IF (MaquinaModoManual) THEN
	//Controle Manual - Válvula Y4
	IF (IhmBt_Y4_Ligar) THEN
		OutValvulaY4R := FALSE;	//Solenóide de Recuo
		OutValvulaY4A := TRUE; //Solenóide de Avanço
	ELSE
		OutValvulaY4A := FALSE;	//Solenóide de Avanço
		OutValvulaY4R := TRUE; //Solenóide de Recuo	
	END_IF
ELSIF (MaquinaModoAuto) THEN
	//Controle Automático - Válvula Y4
	IF (AvancarValvulaY4) THEN
		OutValvulaY4R := FALSE; //Solenóide de Recuo
		OutValvulaY4A := TRUE;	//Solenóide de Avanço
	ELSE
		OutValvulaY4A := FALSE; //Solenóide de Avanço
		OutValvulaY4R := TRUE;	//Solenóide de Recuo
	END_IF
ELSE
	OutValvulaY4R := FALSE; //Solenóide de Recuo
	OutValvulaY4A := FALSE;	//Solenóide de Avanço
END_IF

(*========================================================================*)

(*==============		Válvula Y5 - XXXXXXX XXXXXXX		==============*)

IF (MaquinaModoManual) THEN
	//Controle Manual - Válvula Y5
	IF (IhmBt_Y5_Ligar) THEN
		OutValvulaY5R := FALSE;	//Solenóide de Recuo
		OutValvulaY5A := TRUE; //Solenóide de Avanço
	ELSE
		OutValvulaY5A := FALSE;	//Solenóide de Avanço
		OutValvulaY5R := TRUE; //Solenóide de Recuo	
	END_IF
ELSIF (MaquinaModoAuto) THEN
	//Controle Automático - Válvula Y5
	IF (AvancarValvulaY5) THEN
		OutValvulaY5R := FALSE; //Solenóide de Recuo
		OutValvulaY5A := TRUE;	//Solenóide de Avanço
	ELSE
		OutValvulaY5A := FALSE; //Solenóide de Avanço
		OutValvulaY5R := TRUE;	//Solenóide de Recuo
	END_IF
ELSE
	OutValvulaY5R := FALSE; //Solenóide de Recuo
	OutValvulaY5A := FALSE;	//Solenóide de Avanço
END_IF

(*========================================================================*)

(*==============		Válvula Y6 - XXXXXXX XXXXXXX		==============*)

IF (MaquinaModoManual) THEN
	//Controle Manual - Válvula Y6
	IF (IhmBt_Y6_Ligar) THEN
		OutValvulaY6 := TRUE;
	ELSE
		OutValvulaY6 := FALSE;
	END_IF
ELSIF (MaquinaModoAuto) THEN
	//Controle Automático - Válvula Y6
	IF (LigarValvulaY6) THEN
		OutValvulaY6 := TRUE;
	ELSE
		OutValvulaY6 := FALSE;
	END_IF
ELSE
	OutValvulaY6 := FALSE;
END_IF

(*========================================================================*)

(*==============		Válvula Y9 - XXXXXXX XXXXXXX		==============*)

IF (MaquinaModoManual) THEN
	//Controle Manual - Válvula Y9
	IF (IhmBt_Y9_Ligar) THEN
		OutValvulaY9 := TRUE;
	ELSE
		OutValvulaY9 := FALSE;
	END_IF
ELSIF (MaquinaModoAuto) THEN
	//Controle Automático - Válvula Y9
	IF (LigarValvulaY9) THEN
		OutValvulaY9 := TRUE;
	ELSE
		OutValvulaY9 := FALSE;
	END_IF
ELSE
	OutValvulaY9 := FALSE;
END_IF

(*========================================================================*)

(*==========		Válvula Proporcional - XXXXXXX XXXXXXX		==========*)

IF (MaquinaModoManual) THEN
	//Controle Manual - Válvula Proporcional
	IF (IhmBt_VP_Teste) THEN
		ValvulaProporcional := (INT_TO_REAL(IhmEscr_ValvulaProporcional)/100)*(32767);
	END_IF
ELSIF (MaquinaModoAuto) THEN
	//Controle Automático - Válvula Proporcional
	ValvulaProporcional := (INT_TO_REAL(50)/100)*(32767);
ELSE
	ValvulaProporcional := 0;
END_IF
	
(*========================================================================*)

(*=============		Válvula Y7 - Válvula de Segurança 1		==============*)

//Controle Automático - Válvula Y7
IF (NOT Alarmes.AlarmeGrave) THEN
	LigarValvulaY7 := TRUE;
ELSE
	LigarValvulaY7 := FALSE;
END_IF

//Válvula Y7 - XXXXX XXXXX
IF (LigarValvulaY7) THEN
	OutValvulaY7 := TRUE;
ELSE
	OutValvulaY7 := FALSE;
END_IF

(*========================================================================*) 

(*=============		Válvula Y8 - Válvula de Segurança 2		==============*)

//Controle Automático - Válvula Y8
IF (NOT Alarmes.AlarmeGrave) THEN
	LigarValvulaY8 := TRUE;
ELSE
	LigarValvulaY8 := FALSE;
END_IF

//Válvula Y8 - XXXXX XXXXX
IF (LigarValvulaY8) THEN
	OutValvulaY8 := TRUE;
ELSE
	OutValvulaY8 := FALSE;
END_IF

(*========================================================================*)

END_PROGRAM

// ---- POUs/Perifericos/ReguaPotenciometrica.TcPOU
PROGRAM ReguaPotenciometrica
VAR
	
(*==================		RÉGUA POTENCIOMÉTRICA		==================*)	
 

 
(*========================================================================*)

END_VAR

(*==========		Régua Potênciométrica - EL3004 - 15 bits	==========*)

ReguaPotenciometricaPosicao := (INT_TO_REAL(ReguaPotenciometricaSinal)/32787)*100;

(*=========================		Calibração		==========================*)

IF (MaquinaModoManual) THEN

	IF (IhmBt_ReguaPotenciometrica_CalibrarRecuo) THEN
		ReguaPotenciometrica_Recuada := (INT_TO_REAL(ReguaPotenciometricaSinal)/32787)*100;
		ReguaPotenciometrica_Recuada_LI := (1-(IhmEscr_ReguaPotenciometrica_ToleranciaRecuo/100))*ReguaPotenciometrica_Recuada;
		ReguaPotenciometrica_Recuada_LS := (1+(IhmEscr_ReguaPotenciometrica_ToleranciaRecuo/100))*ReguaPotenciometrica_Recuada;
	END_IF
	
	IF (IhmBt_ReguaPotenciometrica_CalibrarPorca) THEN
		ReguaPotenciometrica_Porca := (INT_TO_REAL(ReguaPotenciometricaSinal)/32787)*100;
		ReguaPotenciometrica_Porca_LI := (1-(IhmEscr_ReguaPotenciometrica_ToleranciaPorca/100))*ReguaPotenciometrica_Porca;
		ReguaPotenciometrica_Porca_LS := (1+(IhmEscr_ReguaPotenciometrica_ToleranciaPorca/100))*ReguaPotenciometrica_Porca;
	END_IF
	
	IF (IhmBt_ReguaPotenciometrica_CalibrarAvanco) THEN
		ReguaPotenciometrica_Avancada := (INT_TO_REAL(ReguaPotenciometricaSinal)/32787)*100;
		ReguaPotenciometrica_Avancada_LI := (1-(IhmEscr_ReguaPotenciometrica_ToleranciaAvanco/100))*ReguaPotenciometrica_Avancada;
		ReguaPotenciometrica_Avancada_LS := (1+(IhmEscr_ReguaPotenciometrica_ToleranciaAvanco/100))*ReguaPotenciometrica_Avancada;
	END_IF
	
END_IF

(*======================		Modo Automático		======================*)


(*========================================================================*)

END_PROGRAM

// ---- POUs/Perifericos/Servos.TcPOU
PROGRAM Servos
VAR
	DelayTeste				: TON;
	
	VetorPosicaoX	: ARRAY[0..15] OF LREAL;
	VetorPosicaoY	: ARRAY[0..15] OF LREAL;
	
	Delay_BtReferenciarServoX 	: TON;
	Delay_BtReferenciarServoY 	: TON;
	
	ServoX_Referenciar			: BOOL;
	ServoY_Referenciar			: BOOL;
	
	ServoX_ReferenciarAuto		: BOOL;
	ServoY_ReferenciarAuto		: BOOL;
	
(*==========================		POWER		==========================*)	

	EixoX_Power 			: MC_Power;	
	EixoX_Power_Busy		: BOOL;
	EixoX_Power_Active		: BOOL;
	EixoX_Power_Error		: BOOL;
	EixoX_Power_ErrorID		: UDINT;
	
	EixoY_Power 			: MC_Power;	
	EixoY_Power_Busy		: BOOL;
	EixoY_Power_Active		: BOOL;
	EixoY_Power_Error		: BOOL;
	EixoY_Power_ErrorID		: UDINT;

(*========================================================================*)

(*==========================		RESET		==========================*)	

	EixoX_Reset 			: MC_Reset;
	EixoX_Reset_Done		: BOOL;	
	EixoX_Reset_Busy		: BOOL;
	EixoX_Reset_Error		: BOOL;
	EixoX_Reset_ErrorID		: UDINT;
	
	EixoY_Reset 			: MC_Reset;
	EixoY_Reset_Done		: BOOL;	
	EixoY_Reset_Busy		: BOOL;
	Eixoy_Reset_Error		: BOOL;
	EixoY_Reset_ErrorID		: UDINT;

(*========================================================================*)

(*==========================		HOME		==========================*)	

	EixoX_Home 						: MC_Home;
	EixoX_Home_Done					: BOOL;	
	EixoX_Home_CommandAborted		: BOOL;
	EixoX_Home_Error				: BOOL;
	EixoX_Home_ErrorID				: UDINT;
	
	HomingMode     					: MC_HomingMode;
	
	EixoY_Home 						: MC_Home;
	EixoY_Home_Done					: BOOL;	
	EixoY_Home_CommandAborted		: BOOL;
	EixoY_Home_Error				: BOOL;
	EixoY_Home_ErrorID				: UDINT;

(*========================================================================*)

(*======================		MOVE ABSOLUTE		======================*)	

	EixoX_MoveAbsHome					: MC_MoveAbsolute;
	EixoX_MoveAbsHome_Done				: BOOL;	
	EixoX_MoveAbsHome_CommandAborted	: BOOL;
	EixoX_MoveAbsHome_Error				: BOOL;
	EixoX_MoveAbsHome_ErrorID			: UDINT;
	
	EixoY_MoveAbsHome					: MC_MoveAbsolute;
	EixoY_MoveAbsHome_Done				: BOOL;	
	EixoY_MoveAbsHome_CommandAborted	: BOOL;
	EixoY_MoveAbsHome_Error				: BOOL;
	EixoY_MoveAbsHome_ErrorID			: UDINT;

	EixoX_MoveAbsolute 					: MC_MoveAbsolute;
	EixoX_MoveAbsolute_Done				: BOOL;	
	EixoX_MoveAbsolute_CommandAborted	: BOOL;
	EixoX_MoveAbsolute_Error			: BOOL;
	EixoX_MoveAbsolute_ErrorID			: UDINT;
	
	EixoY_MoveAbsolute			 		: MC_MoveAbsolute;
	EixoY_MoveAbsolute_Done				: BOOL;	
	EixoY_MoveAbsolute_CommandAborted	: BOOL;
	EixoY_MoveAbsolute_Error			: BOOL;
	EixoY_MoveAbsolute_ErrorID			: UDINT;

(*========================================================================*)
	
(*=========================		MOVE JOG		==========================*)	

	EixoX_MoveJog					: MC_Jog;
	EixoY_MoveJog					: MC_Jog;
	
	EixoX_JogReferenciarAuto		: MC_Jog;
	EixoY_JogReferenciarAuto		: MC_Jog;
	
(*========================================================================*)	

(*======================		MOVE RELATIVE		======================*)	

	EixoX_MoveRelative		: MC_MoveRelative;
	EixoY_MoveRelative		: MC_MoveRelative;

(*========================================================================*)

(*=====================		MÁQUINA DE ESTADOS		======================*)	

	PassoServosXY				: INT;
	index						: INT;
	PosicaoX					: LREAL;
	PosicaoY					: LREAL;
	
	Flag_EixoX_PosicaoOK		: BOOL;
	Flag_EixoY_PosicaoOK		: BOOL;
	
	PassoEixoXReferenciarAutoINICIO	: INT;
	PassoEixoXReferenciarAutoFIM	: INT;
	PassoEixoYReferenciarAutoINICIO	: INT;
	PassoEixoYReferenciarAutoFIM	: INT;
	
	JogFwd_EixoX_ReferenciarAuto	: BOOL;
	JogBwd_EixoX_ReferenciarAuto	: BOOL;

	JogFwd_EixoY_ReferenciarAuto	: BOOL;
	JogBwd_EixoY_ReferenciarAuto	: BOOL;

(*========================================================================*)
	
	//Blocos de Controle Eixo X
	PowerOnServoX		: BOOL;
	ReferenciarServoX	: BOOL;
	MoveHomeServoX		: BOOL;
	ResetServoX			: BOOL;
	JogFwdServoX		: BOOL;
	JogBwdServoX		: BOOL;
	
	//Status Servo Eixo X
	VelocidadeEixoX		: LREAL;
	PosicaoEixoX		: LREAL;
	TorqueEixoX			: LREAL;
	
	//Blocos de Controle Eixo Y
	PowerOnServoY		: BOOL;
	ReferenciarServoY	: BOOL;
	MoveHomeServoY		: BOOL;
	ResetServoY			: BOOL;
	JogFwdServoY		: BOOL;
	JogBwdServoY		: BOOL;
	
	//Status Servo Eixo X
	VelocidadeEixoY		: LREAL;
	PosicaoEixoY		: LREAL;
	TorqueEixoY			: LREAL;
	
END_VAR

IhmEscr_ServoXY_VelocidadeManual := 5;

(*=================		POWER - SERVOS EIXOS X E Y		==================*)

(*======================		SERVO EIXO X		======================*)

EixoX_Power_Busy 	:= EixoX_Power.Busy;
EixoX_Power_Active 	:= EixoX_Power.Active;
EixoX_Power_Error 	:= EixoX_Power.Error;
EixoX_Power_ErrorID	:= EixoX_Power.ErrorID;

IF (MaquinaModoManual AND NOT Alarmes.AlarmeGrave)THEN
	EixoX_Power(Axis := EixoX,
				Enable := IhmBt_ServoX_PowerOn,
				Enable_Positive := IhmBt_ServoX_PowerOn,
				Enable_Negative := IhmBt_ServoX_PowerOn,
				Override := 100);
ELSIF (NOT Alarmes.AlarmeGrave) THEN
	EixoX_Power(Axis := EixoX,
			Enable := TRUE,
			Enable_Positive := TRUE,
			Enable_Negative := TRUE,
			Override := 100);
ELSE
	EixoX_Power(Axis := EixoX,
			Enable := FALSE,
			Enable_Positive := FALSE,
			Enable_Negative := FALSE);
END_IF
				
IF EixoX_Power.Status THEN
	EixoX_Energizado := TRUE;
ELSE
	EixoX_Energizado := FALSE;
END_IF

(*======================		SERVO EIXO Y		======================*)

EixoY_Power_Busy 	:= EixoY_Power.Busy;
EixoY_Power_Active 	:= EixoY_Power.Active;
EixoY_Power_Error 	:= EixoY_Power.Error;
EixoY_Power_ErrorID	:= EixoY_Power.ErrorID;

IF (MaquinaModoManual AND NOT Alarmes.AlarmeGrave)THEN
	EixoY_Power(Axis := EixoY,
				Enable := IhmBt_ServoY_PowerOn,
				Enable_Positive := IhmBt_ServoY_PowerOn,
				Enable_Negative := IhmBt_ServoY_PowerOn,
				Override := 100);
ELSIF (NOT Alarmes.AlarmeGrave) THEN
	EixoY_Power(Axis := EixoY,
			Enable := TRUE,
			Enable_Positive := TRUE,
			Enable_Negative := TRUE,
			Override := 100);
ELSE
	EixoY_Power(Axis := EixoY,
			Enable := FALSE,
			Enable_Positive := FALSE,
			Enable_Negative := FALSE);
END_IF
			
IF EixoY_Power.Status THEN
	EixoY_Energizado := TRUE;
ELSE
	EixoY_Energizado := FALSE;
END_IF

(*=================		RESET - SERVOS EIXOS X E Y		==================*)

(*======================		SERVO EIXO X		======================*)

EixoX_Reset_Done 	:= EixoX_Reset.Done;
EixoX_Reset_Busy 	:= EixoX_Reset.Busy;
EixoX_Reset_Error 	:= EixoX_Reset.Error;
EixoX_Reset_ErrorID	:= EixoX_Reset.ErrorID;

EixoX_Reset(Axis := EixoX, Execute := (IhmBt_ServoX_Reset OR Reset));

(*======================		SERVO EIXO Y		======================*)

EixoY_Reset_Done 	:= EixoY_Reset.Done;
EixoY_Reset_Busy 	:= EixoY_Reset.Busy;
EixoY_Reset_Error 	:= EixoY_Reset.Error;
EixoY_Reset_ErrorID	:= EixoY_Reset.ErrorID;

EixoY_Reset(Axis := EixoY, Execute := (IhmBt_ServoX_Reset OR Reset));

(*=============		REFERENCIAR - SERVOS EIXOS X E Y		==============*)

(*======================		SERVO EIXO X		======================*)

EixoX_Home_Done 			:= EixoX_Home.Done;
EixoX_Home_CommandAborted 	:= EixoX_Home.CommandAborted;
EixoX_Home_Error 			:= EixoX_Home.Error;
EixoX_Home_ErrorID			:= EixoX_Home.ErrorID;

//Lógica para Delay ao pressionar o botão de referenciar
	IF (IhmBt_ServoX_Referenciar) THEN
		Delay_BtReferenciarServoX(IN := TRUE, PT := T#2S);
		IF(Delay_BtReferenciarServoX.Q) THEN
			ServoX_Referenciar := TRUE;
		END_IF
	ELSE
		Delay_BtReferenciarServoX(IN := FALSE);
		ServoX_Referenciar := FALSE;
	END_IF

EixoX_Home(Axis := EixoX, Position := 0, HomingMode := MC_Direct, Execute := ((ServoX_Referenciar AND MaquinaModoManual) OR ServoX_ReferenciarAuto));

(*======================		SERVO EIXO Y		======================*)

EixoY_Home_Done 			:= EixoY_Home.Done;
EixoY_Home_CommandAborted 	:= EixoY_Home.CommandAborted;
EixoY_Home_Error 			:= EixoY_Home.Error;
EixoY_Home_ErrorID			:= EixoY_Home.ErrorID;

//Lógica para Delay ao pressionar o botão de referenciar
	IF (IhmBt_ServoY_Referenciar) THEN
		Delay_BtReferenciarServoY(IN := TRUE, PT := T#2S);
		IF(Delay_BtReferenciarServoY.Q) THEN
			ServoY_Referenciar := TRUE;
		END_IF
	ELSE
		Delay_BtReferenciarServoY(IN := FALSE);
		ServoY_Referenciar := FALSE;
	END_IF

EixoY_Home(Axis := EixoY, Position := 0, HomingMode := MC_Direct, Execute := ((ServoY_Referenciar AND MaquinaModoManual) OR ServoY_ReferenciarAuto));

(*=============		MOVE para HOME - SERVOS EIXOS X E Y		==============*)

(*======================		SERVO EIXO X		======================*)

EixoX_MoveAbsHome(	Axis := EixoX,
					Execute := (IhmBt_ServoX_Home AND MaquinaModoManual),
					Position := 0,
					Velocity := IhmEscr_ServoXY_VelocidadeAuto
					(*Direction := 2*));

(*======================		SERVO EIXO Y		======================*)
								
EixoX_MoveAbsHome(	Axis := EixoY,
					Execute := (IhmBt_ServoY_Home AND MaquinaModoManual),
					Position := 0,
					Velocity := IhmEscr_ServoXY_VelocidadeAuto
					(*Direction := 2*));

(*=================		MANUAL - SERVOS EIXOS X E Y		==================*)

(*======================		SERVO EIXO X		======================*)

EixoX_MoveJog(	Axis := EixoX,
				JogForward := (IhmBt_ServoX_JogFwd AND MaquinaModoManual),
				JogBackwards := (IhmBt_ServoX_JogBwd AND MaquinaModoManual),
				Velocity := IhmEscr_ServoXY_VelocidadeManual,
				Acceleration := 100,
				Deceleration := 100);
				
(*======================		SERVO EIXO Y		======================*)
								
EixoY_MoveJog(	Axis := EixoY,
				JogForward := (IhmBt_ServoY_JogFwd AND MaquinaModoManual),
				JogBackwards := (IhmBt_ServoY_JogBwd AND MaquinaModoManual),
				Velocity := IhmEscr_ServoXY_VelocidadeManual,
				Acceleration := 100,
				Deceleration := 100);

(*=================		STATUS - SERVOS EIXOS X E Y		==================*)

(*======================		SERVO EIXO X		======================*)

IhmLeit_ServoX_Posicao		:= EixoX.NcToPlc.ActPos;
IhmLeit_ServoX_Velocidade	:= EixoX.NcToPlc.ActVelo;
IhmLeit_ServoX_Torque		:= EixoX.NcToPlc.ActTorque;

(*======================		SERVO EIXO Y		======================*)

IhmLeit_ServoY_Posicao		:= EixoY.NcToPlc.ActPos;
IhmLeit_ServoY_Velocidade	:= EixoY.NcToPlc.ActVelo;
IhmLeit_ServoY_Torque		:= EixoY.NcToPlc.ActTorque;

(*=========		MANIVELA ELETRÔNICA - SERVOS EIXOS X E Y		==========*)



(*=================		AUTOMÁTICO - SERVOS EIXOS X E Y		==============*)
(*======================		Modo Automático		======================*)

//Receita Teste

PosicaoOrigemX := 20;
PosicaoOrigemY := 31;

VetorPosicaoX[0] := 20;
VetorPosicaoY[0] := 31;

VetorPosicaoX[1] := 59;
VetorPosicaoY[1] := 15;

//PosicaoOrigemX := TargetX[0];
//PosicaoOrigemY := TargetY[0];

//Condição de Bloqueio da Máquina de Estados - Servos XY
IF (Alarmes.AlarmeGrave
	//OR NOT Alarmes.AlarmeMedio
	OR NOT MaquinaLigada
	OR NOT MaquinaModoAuto
	//OR NOT((ReguaPotenciometricaPosicao > ReguaPotenciometrica_Recuada_LI) AND (ReguaPotenciometricaPosicao < ReguaPotenciometrica_Recuada_LS))
	) THEN
	PassoServosXY := 1000;
	Flag_ServosXY_Maquina := FALSE;
	index := 0;
	EixoX_MoveAbsolute(	Axis:= EixoX, Execute:= FALSE);
	EixoY_MoveAbsolute(	Axis:= EixoY, Execute:= FALSE);
	Flag_EixoX_PosicaoOK := FALSE;
	Flag_EixoY_PosicaoOK := FALSE;
	
END_IF

CASE PassoServosXY OF
	
	//Passo 0 - Inicialização	
	0: PassoServosXY := 10;
		
	//Passo 10 - Condição para Iniciar a Rotina dos Servos XY
	10: IF  (Flag_Maquina_ServosXY) THEN
			Flag_Maquina_ServosXY := FALSE;
			PassoServosXY := 20;
		END_IF
		
	//Passo 20 - Soldar 
	20:	IF (TRUE OR SoldaXY[index]) THEN
			Flag_ServosXY_MaquinaSolda := TRUE;
			PassoServosXY := 30;
		ELSE
			Flag_ServosXY_MaquinaSolda := FALSE;
			PassoServosXY := 40;			
		END_IF

	//Passo 30 - Aguardar conclusão de Solda
	30:	IF (Flag_MaquinaSolda_ServosXY) THEN
			Flag_MaquinaSolda_ServosXY := FALSE;
			PassoServosXY := 40;			
		END_IF
	
	//Passo 40 - Validar Próximo Ponto (X,Y)
	40: index := index + 1;
		IF (index<=(NumPontosSolda-1)) THEN
			PassoServosXY := 50;	
		ELSE
			index := 0;
			PassoServosXY := 80;	
		END_IF
	
	//Passo 50 - Carregar Posição Alvo - Servo X e Y 
	50: PosicaoX := VetorPosicaoX[index];//TargetX[index];
		PosicaoY := VetorPosicaoY[index];//TargetY[index];
		PassoServosXY := 60;
		
	//Passo 60 - Movimentar Servo Eixos X e Y
	//			aguardar conclusão do movimento
	60: EixoX_MoveAbsolute(	Axis:= EixoX, 
							Execute:= TRUE,
							Position:= PosicaoX,
							Velocity:= IhmEscr_ServoXY_VelocidadeAuto
							//Acceleration:= 15000,
							//Deceleration:= 15000
							);			
		IF (EixoX_MoveAbsolute.Done) THEN
			Flag_EixoX_PosicaoOK := TRUE;
		END_IF
							
		EixoY_MoveAbsolute(	Axis:= EixoY, 
							Execute:= TRUE,
							Position:= PosicaoY,
							Velocity:= IhmEscr_ServoXY_VelocidadeAuto
							//Acceleration:= 15000,
							//Deceleration:= 15000
							);
		IF (EixoY_MoveAbsolute.Done) THEN
			Flag_EixoY_PosicaoOK := TRUE;	
		END_IF
		
		IF (Flag_EixoX_PosicaoOK AND Flag_EixoY_PosicaoOK) THEN
			PassoServosXY := 70;	
		END_IF
		
	//Passo 70 - Finalizar Movimentação - Servos X e Y
	70: EixoX_MoveAbsolute(	Axis:= EixoX, Execute:= FALSE);
		EixoY_MoveAbsolute(	Axis:= EixoY, Execute:= FALSE);
		Flag_EixoX_PosicaoOK := FALSE;
		Flag_EixoY_PosicaoOK := FALSE;
		PassoServosXY := 75;
		
	//Passo 75 - Aguardar Delay de Teste
	75: DelayTeste(IN:=TRUE,PT:=T#200MS);
		IF DelayTeste.Q THEN
			DelayTeste(IN:=FALSE);
			PassoServosXY := 20;		
		END_IF
		
	//Passo 80 - Movimentar Servos X e  para a Origem
	//			e aguardar conclusão do movimento
	80: EixoX_MoveAbsolute(	Axis := EixoX, 
							Execute := TRUE,
							Position := VetorPosicaoX[0],
							Velocity := IhmEscr_ServoXY_VelocidadeAuto
							//Acceleration:= 15000,
							//Deceleration:= 15000
							);
		IF (EixoX_MoveAbsolute.Done) THEN
			Flag_EixoX_PosicaoOK := TRUE;	
		END_IF
		
		EixoY_MoveAbsolute(	Axis := EixoY, 
							Execute := TRUE,
							Position := VetorPosicaoY[0],
							Velocity := IhmEscr_ServoXY_VelocidadeAuto
							//Acceleration:= 15000,
							//Deceleration:= 15000
							);
		IF (EixoY_MoveAbsolute.Done) THEN
			Flag_EixoY_PosicaoOK := TRUE;	
		END_IF
		
		IF (Flag_EixoX_PosicaoOK AND Flag_EixoY_PosicaoOK) THEN
			PassoServosXY := 90;	
		END_IF
		
	//Passo 90 - Finalizar Movimentação - Servos X e Y
	90: EixoX_MoveAbsolute(	Axis:= EixoX, Execute:= FALSE);
		EixoY_MoveAbsolute(	Axis:= EixoY, Execute:= FALSE);
		Flag_EixoX_PosicaoOK := FALSE;
		Flag_EixoY_PosicaoOK := FALSE;
		PassoServosXY := 100;
		
	//Passo 100 - Sinalizar Conclusão da Rotina
	100:	Flag_ServosXY_Maquina := TRUE;
		PassoServosXY := 1000;

	//Passo 1000 - Finalização
	1000: PassoServosXY := 0;
	
END_CASE

(*=================		REFERENCIAMENTO AUTOMÁTICO		==================*)

(*======================		SERVO EIXO X		======================*)
								
EixoX_JogReferenciarAuto(	Axis := EixoX,
							JogForward := (JogFwd_EixoX_ReferenciarAuto),
							JogBackwards := (JogBwd_EixoX_ReferenciarAuto),
							Velocity := 1,
							Acceleration := 100,
							Deceleration := 100);
							
//Condição de Bloqueio da Máquina de Estados - Referenciamento Auto (INICIO)
IF (Alarmes.AlarmeGrave
	OR MaquinaLigada
	OR NOT MaquinaModoManual
	OR NOT IhmBt_ServoX_ReferenciarAutoINICIO
	OR	IhmBt_ServoX_ReferenciarAutoFIM
	OR NOT IhmBt_ServoX_PowerOn
	OR InFimCurso3
	) THEN
	PassoEixoXReferenciarAutoINICIO := 1000;
	//JogFwd_EixoX_ReferenciarAuto := FALSE;
	JogBwd_EixoX_ReferenciarAuto := FALSE;
	//ServoX_ReferenciarAuto := FALSE;
END_IF

CASE PassoEixoXReferenciarAutoINICIO OF

	//Passo 0 - Inicialização
	0: PassoEixoXReferenciarAutoINICIO := 10;
	
	//Passo 10 - Condição para iniciar Rotina de Referenciamento Automático
	10: IF (IhmBt_ServoX_ReferenciarAutoINICIO) THEN
			PassoEixoXReferenciarAutoINICIO := 20;
		END_IF
		
	//Passo 20 - Move Jog BWD - Referenciar 
	20: JogBwd_EixoX_ReferenciarAuto := TRUE;
		PassoEixoXReferenciarAutoINICIO := 30;

	//Passo 30 - Aguardar Acionamento do Switch Fim de Curso
	30: IF (InFimCurso3) THEN
			JogBwd_EixoX_ReferenciarAuto := TRUE;
			//ServoX_ReferenciarAuto := TRUE;
			PassoEixoXReferenciarAutoINICIO := 40;
		END_IF
		
	//Passo 40 - Sinalizar Conclusão da Rotina
	40: IhmBt_ServoX_ReferenciarAutoINICIO := FALSE;
		//ServoX_ReferenciarAuto := FALSE;
		PassoEixoXReferenciarAutoINICIO := 1000;
	
	//Passo 1000 - Finalização
	1000:	IhmBt_ServoX_ReferenciarAutoINICIO := FALSE;
			PassoEixoXReferenciarAutoINICIO := 0;

END_CASE

//Condição de Bloqueio da Máquina de Estados - Referenciamento Auto (FIM)
IF (Alarmes.AlarmeGrave
	OR MaquinaLigada
	OR NOT MaquinaModoManual
	OR NOT IhmBt_ServoX_ReferenciarAutoFIM
	OR IhmBt_ServoX_ReferenciarAutoINICIO
	OR NOT IhmBt_ServoX_PowerOn
	OR InFimCurso4
	) THEN
	PassoEixoXReferenciarAutoFIM := 1000;
	JogFwd_EixoX_ReferenciarAuto := FALSE;
	//JogBwd_EixoX_ReferenciarAuto := FALSE;
	//ServoX_ReferenciarAuto := FALSE;
END_IF

CASE PassoEixoXReferenciarAutoFIM OF

	//Passo 0 - Inicialização
	0: PassoEixoXReferenciarAutoFIM := 10;
	
	//Passo 10 - Condição para iniciar Rotina de Referenciamento Automático
	10: IF (IhmBt_ServoX_ReferenciarAutoFIM) THEN
			PassoEixoXReferenciarAutoFIM := 20;
		END_IF
		
	//Passo 20 - Move Jog FWD - Referenciar 
	20: JogFwd_EixoX_ReferenciarAuto := TRUE;
		PassoEixoXReferenciarAutoFIM := 30;

	//Passo 30 - Aguardar Acionamento do Switch Fim de Curso
	30: IF (InFimCurso4) THEN
			JogFwd_EixoX_ReferenciarAuto := TRUE;
			//ServoX_ReferenciarAuto := TRUE;
			PassoEixoXReferenciarAutoFIM := 40;
		END_IF
		
	//Passo 40 - Sinalizar Conclusão da Rotina
	40: IhmBt_ServoX_ReferenciarAutoFIM := FALSE;
		//ServoX_ReferenciarAuto := FALSE;
		PassoEixoXReferenciarAutoFIM := 1000;
	
	//Passo 1000 - Finalização
	1000:	IhmBt_ServoX_ReferenciarAutoFIM := FALSE;
			PassoEixoXReferenciarAutoFIM := 0;

END_CASE

(*======================		SERVO EIXO Y		======================*)
								
EixoY_JogReferenciarAuto(	Axis := EixoY,
							JogForward := (JogFwd_EixoY_ReferenciarAuto),
							JogBackwards := (JogBwd_EixoY_ReferenciarAuto),
							Velocity := 1,
							Acceleration := 100,
							Deceleration := 100);
							
//Condição de Bloqueio da Máquina de Estados - Referenciamento Auto (INICIO)
IF (Alarmes.AlarmeGrave
	OR MaquinaLigada
	OR NOT MaquinaModoManual
	OR NOT IhmBt_ServoY_ReferenciarAutoINICIO
	OR IhmBt_ServoY_ReferenciarAutoFIM
	OR NOT IhmBt_ServoY_PowerOn
	OR InFimCurso1
	) THEN
	PassoEixoYReferenciarAutoINICIO := 1000;
	//JogFwd_EixoY_ReferenciarAuto := FALSE;
	JogBwd_EixoY_ReferenciarAuto := FALSE;
	//ServoY_ReferenciarAuto := FALSE;
END_IF

CASE PassoEixoYReferenciarAutoINICIO OF

	//Passo 0 - Inicialização
	0: PassoEixoYReferenciarAutoINICIO := 10;
	
	//Passo 10 - Condição para iniciar Rotina de Referenciamento Automático
	10: IF (IhmBt_ServoY_ReferenciarAutoINICIO) THEN
			PassoEixoYReferenciarAutoINICIO := 20;
		END_IF
		
	//Passo 20 - Move Jog BWD - Referenciar 
	20: JogBwd_EixoY_ReferenciarAuto := TRUE;
		PassoEixoYReferenciarAutoINICIO := 30;

	//Passo 30 - Aguardar Acionamento do Switch Fim de Curso
	30: IF (InFimCurso1) THEN
			JogBwd_EixoY_ReferenciarAuto := TRUE;
			//ServoY_ReferenciarAuto := TRUE;
			PassoEixoYReferenciarAutoINICIO := 40;
		END_IF
		
	//Passo 40 - Sinalizar Conclusão da Rotina
	40: IhmBt_ServoY_ReferenciarAutoINICIO := FALSE;
		//ServoY_ReferenciarAuto := FALSE;
		PassoEixoYReferenciarAutoINICIO := 1000;
	
	//Passo 1000 - Finalização
	1000:	IhmBt_ServoY_ReferenciarAutoINICIO := FALSE;
			PassoEixoYReferenciarAutoINICIO := 0;

END_CASE

//Condição de Bloqueio da Máquina de Estados - Referenciamento Auto (FIM)
IF (Alarmes.AlarmeGrave
	OR MaquinaLigada
	OR NOT MaquinaModoManual
	OR NOT IhmBt_ServoY_ReferenciarAutoFIM
	OR IhmBt_ServoY_ReferenciarAutoINICIO
	OR NOT IhmBt_ServoY_PowerOn
	OR InFimCurso2
	) THEN
	PassoEixoYReferenciarAutoFIM := 1000;
	JogFwd_EixoY_ReferenciarAuto := FALSE;
	//JogBwd_EixoY_ReferenciarAuto := FALSE;
	//ServoY_ReferenciarAuto := FALSE;
END_IF

CASE PassoEixoYReferenciarAutoFIM OF

	//Passo 0 - Inicialização
	0: PassoEixoYReferenciarAutoFIM := 10;
	
	//Passo 10 - Condição para iniciar Rotina de Referenciamento Automático
	10: IF (IhmBt_ServoY_ReferenciarAutoFIM) THEN
			PassoEixoYReferenciarAutoFIM := 20;
		END_IF
		
	//Passo 20 - Move Jog FWD - Referenciar 
	20: JogBwd_EixoY_ReferenciarAuto := TRUE;
		PassoEixoYReferenciarAutoFIM := 30;

	//Passo 30 - Aguardar Acionamento do Switch Fim de Curso
	30: IF (InFimCurso1) THEN
			JogBwd_EixoY_ReferenciarAuto := TRUE;
			//ServoY_ReferenciarAuto := TRUE;
			PassoEixoYReferenciarAutoFIM := 40;
		END_IF
		
	//Passo 40 - Sinalizar Conclusão da Rotina
	40: IhmBt_ServoY_ReferenciarAutoFIM := FALSE;
		//ServoY_ReferenciarAuto := FALSE;
		PassoEixoYReferenciarAutoFIM := 1000;
	
	//Passo 1000 - Finalização
	1000:	IhmBt_ServoY_ReferenciarAutoFIM := FALSE;
			PassoEixoYReferenciarAutoFIM := 0;

END_CASE

(*========================================================================*)

END_PROGRAM

// ---- POUs/Perifericos/Robo.TcPOU
PROGRAM Robo
VAR

	BT_test						: BOOL;
	TON_DelayTesteExpPeca		: TON;
	
	//index						: INT;

(*=====================		ROBO YASKAWA		==========================*)	
 
 PassoRoboAuto				: INT;
 
 Flag_PLC_Robot_WorkHome		: BOOL; //Retonar a para a posição WORK HOME (Ordem PLC)
 Flag_PLC_Robot_PegarPeca		: BOOL; //Pegar Peça na Mesa Indexadora (Ordem PLC)
 Flag_PLC_Robot_Camera			: BOOL; //Levar Peça Até a Câmera (Ordem PLC)
 Flag_PLC_Robot_CapturarImagens	: BOOL;
 Flag_PLC_Robot_Aprovada		: BOOL; //Levar Peça Até a Caixa - Aprovada (Ordem PLC)
 Flag_PLC_Robot_Reprovada		: BOOL; //Descartar Peça (Ordem PLC)
 
 Flag_Robot_PLC_WorkHome		: BOOL; //Retonar a para a posição WORK HOME (Conclusão Robô)
 Flag_Robot_PLC_PegarPeca		: BOOL; //Pegar Peça na Mesa Indexadora (Conclusão Robô)
 Flag_Robot_PLC_Camera			: BOOL; //Levar Peça Até a Câmera (Conclusão Robô)
 Flag_Robot_PLC_CapturarImagens	: BOOL;
 Flag_Robot_PLC_Aprovada		: BOOL; //Levar Peça Até a Caixa - Aprovada (Conclusão Robô)
 Flag_Robot_PLC_Reprovada		: BOOL; //Descartar Peça (Conclusão Robô)

(*========================================================================*)

END_VAR

(*==========		Robô Yaskawa Comunicação Ethernet/IP		==========*)

//PLC to Robot -> Byte 0

PLC_Robot_0.0 := Robot_CallMasterJob;
PLC_Robot_0.1 := Robot_ServoOn;
PLC_Robot_0.2 := Robot_ServoOff;
PLC_Robot_0.3 := Robot_ExtStart;
PLC_Robot_0.4 := Robot_ResetAlarm;

//PLC_Robot_0.4 := Robot_JobBegin;

//PLC to Robot -> Byte 1

PLC_Robot_1.0 := Robot_JobCamera;

//PLC to Robot -> Byte 2

PLC_Robot_3 := 1; //Receita



Robot_NotSafetyPosition := Robot_PLC_0.3;
Robot_JobCompleted := Robot_PLC_1.0;

//Robot_Home:= Robot_PLC_1.0;

Robot_Peca	:= Robot_PLC_2.0;
Robot_Foto1	:= Robot_PLC_2.1;
Robot_Foto2	:= Robot_PLC_2.2;


Robot_HomePosition 	:= Robot_PLC_1.0;
Robot_TopMasterJob	:= Robot_PLC_1.1;
Robot_AlarmStatus 	:= Robot_PLC_1.2;




Robot_JobCamera := TRUE;

//Robot_PLC_1.0 := Valvula


(*=========================		Modo Manual		==========================*)

 PLC_Robot_2.0 := Flag_PLC_Robot_PegarPeca;
 PLC_Robot_2.1 := Flag_PLC_Robot_Camera;
 PLC_Robot_2.2 := Flag_PLC_Robot_CapturarImagens;
 PLC_Robot_2.3 := Flag_PLC_Robot_Aprovada;
 PLC_Robot_2.4 := Flag_PLC_Robot_Reprovada;
 PLC_Robot_2.5 := Flag_PLC_Robot_WorkHome;
 
 Flag_Robot_PLC_PegarPeca 		:= Robot_PLC_2.0;
 Flag_Robot_PLC_Camera 			:= Robot_PLC_2.1;
 Flag_Robot_PLC_CapturarImagens := Robot_PLC_2.2;
 Flag_Robot_PLC_Aprovada 		:= Robot_PLC_2.3;
 Flag_Robot_PLC_Reprovada 		:= Robot_PLC_2.4;
 Flag_Robot_PLC_WorkHome 		:= Robot_PLC_2.5;
 
(*======================		Modo Automático		======================*)

//Condição de Bloqueio da Máquina de Estados - Robô Yaskawa
IF (Alarmes.AlarmeGrave
	//OR NOT Alarmes.AlarmeMedio
	//OR NOT MaquinaLigada
	//OR NOT MaquinaModoAuto
	) THEN
	PassoRoboAuto := 1000;
	Camera_indexJob := 0;
END_IF

CASE PassoRoboAuto OF
	
	//Passo 0 - Inicialização	
	0: PassoRoboAuto := 10;
	   
	//Passo 10 - Condição para Iniciar a Rotina do Robo
	10: IF (Flag_Maquina_Robo) THEN
				Flag_Maquina_Robo := FALSE;
			PassoRoboAuto := 20;
		END_IF
		
	//Passo 20 - Verifica Posição do Robo
	20: IF (Robot_HomePosition) THEN
			PassoRoboAuto := 30;
		END_IF
		
	//Passo 30 - Verificar Flag Posição
	30:	IF (Flag_Robot_PLC_WorkHome) THEN
			PassoRoboAuto := 40;
		END_IF
			
	//Passo 40 - Iniciar Ciclo - Pegar Peça no Mesa Index
	40: Flag_PLC_Robot_PegarPeca := TRUE;
		IF (Flag_Robot_PLC_PegarPeca) THEN
			Flag_PLC_Robot_PegarPeca := FALSE;
			PassoRoboAuto := 50;	
		END_IF
		
	//Passo 50 - Levar Peça até a Câmera SICK 
	50: Flag_PLC_Robot_Camera := TRUE;
		IF (Flag_Robot_PLC_Camera) THEN
			Flag_PLC_Robot_Camera := FALSE;
			PassoRoboAuto := 60;	
		END_IF
			
	//Passo 60 - Sinalizar Captura de Imagens
	60: Flag_PLC_Robot_CapturarImagens := TRUE;
		IF (NOT Flag_Robot_PLC_Camera) THEN
			Flag_PLC_Robot_CapturarImagens := FALSE;
			PassoRoboAuto := 70;	
		END_IF
		
	//Passo 70 - Capturar Imagens
	70: Flag_Robo_Camera := TRUE;
		PassoRoboAuto := 80;
	
	//Passo 80 - Aguardar Conclusão da Capturar Imagens
	80: IF (Flag_Camera_Robo) THEN
			Flag_Camera_Robo := FALSE;
			PassoRoboAuto := 90;	
		END_IF	
			
	//Passo 90 - Avaliar Resultado da Câmera
	90: IF(PecaAprovada) THEN
			PecaAprovada := FALSE;
			PassoRoboAuto := 100;
		ELSE
			Camera_indexJob := 0;
			PassoRoboAuto := 120;
		END_IF

	//Passo 100 - Validar próximo ponto	
	100: IF (Camera_indexJob + 1 < NumPontosCamera) THEN
			Camera_indexJob := Camera_indexJob + 1;
			PassoRoboAuto := 50;
		ELSE
			Camera_indexJob := 0;
			PassoRoboAuto := 100;
		END_IF
	
	
	//Passo 100 - Depositar a Peça Aprovada na Caixa 
	110: Flag_PLC_Robot_Aprovada := TRUE;
		IF (Flag_Robot_PLC_Aprovada) THEN
			Flag_PLC_Robot_Aprovada := FALSE;
			
			//Expelir Peça da Garra
			AvancarValvulaY1 := TRUE;
			TON_DelayTesteExpPeca(IN := TRUE, PT := T#3S);
			IF (TON_DelayTesteExpPeca.Q) THEN
				TON_DelayTesteExpPeca(IN := FALSE);
				AvancarValvulaY1 := FALSE;
				PassoRoboAuto := 115;	
			END_IF

		END_IF
	
	//Passo 115 - Atualizar Contador de Peças Aprovadas
	115: Contador_PecasAprovadas := Contador_PecasAprovadas + 1;
		PassoRoboAuto := 130; 
		
	//Passo 120 - Descartar a Peça Reprovada 
	120: Flag_PLC_Robot_Reprovada := TRUE;
		IF (Flag_Robot_PLC_Reprovada) THEN
			Flag_PLC_Robot_Reprovada := FALSE;
			
			//Expelir Peça da Garra
			AvancarValvulaY1 := TRUE;
			TON_DelayTesteExpPeca(IN := TRUE, PT := T#3S);
			IF (TON_DelayTesteExpPeca.Q) THEN
				TON_DelayTesteExpPeca(IN := FALSE);
				AvancarValvulaY1 := FALSE;
				PassoRoboAuto := 125;
			END_IF
			
		END_IF
		
	//Passo 125 - Atualizar Contador de Peças Reprovadas
	125: Contador_PecasReprovadas := Contador_PecasReprovadas + 1;
		PassoRoboAuto := 130; 
	
	//Passo 130 - Atualizar Contador Total
	130: Contador_Total := Contador_PecasAprovadas + Contador_PecasReprovadas;
		PassoRoboAuto := 140; 
	
	//Passo 140 - Retornar a Posição WORK HOME 
	140: Flag_PLC_Robot_WorkHome := TRUE;
		IF (Flag_Robot_PLC_WorkHome) THEN
			Flag_PLC_Robot_WorkHome := FALSE;
			PassoRoboAuto := 150;	
		END_IF
		
	//Passo 150 - Sinalizar Conclusão da Rotina 
	150: Flag_Robo_Maquina := TRUE;
		PassoRoboAuto := 1000;

	//Passo 1000 - Finalização
	1000: PassoRoboAuto := 0;
	
END_CASE

(*========================================================================*)

END_PROGRAM

// ---- POUs/Perifericos/Camera.TcPOU
PROGRAM Camera
VAR

	BT_test						: BOOL;
	
	TON_DelayTest1				: TON;
	TON_DelayTest2				: TON;
	TON_DelayTest3				: TON;
	TON_DelayTest4				: TON;
	TON_DelayTest5				: TON;

(*=========================		CAMERA SICK		==========================*)	
 
 PassoCameraAuto			: INT;
 TON_CameraError			: TON;
 TON_CameraChangeJob		: TON;
 
(*========================================================================*)

END_VAR

(*=============		Câmera Sick Comunicação Ethernet/IP		==============*)

Camera_JobResult := CameraSickIn_3.0;
Camera_JobCompleted := CameraSickIn_0.2;
Camera_JobID := CameraSickIn_2;

CameraSickOut_0.0 := Camera_Trigger;
CameraSickOut_0.1 := Camera_ChangeJob;
CameraSickOut_2 := Camera_SetJob;

(*========================================================================*)

IhmLeit_Camera_JobID := BYTE_TO_INT(Camera_JobID);

IhmVs_Camera_JobResult_Text := 'Test';

(*=========================		Modo Manual		==========================*)

IF (MaquinaModoManual) THEN

	Camera_SetJob := INT_TO_BYTE(IhmEscr_Camera_SetJob);
	Camera_ChangeJob := IhmBt_Camera_ChangeJob;
	Camera_Trigger := IhmBt_Camera_Trigger;

END_IF

(*======================		Modo Automático		======================*)

Camera_TargetJob[0] := 1;
Camera_TargetJob[1] := 2;

//Condição de Bloqueio da Máquina de Estados - Câmera SICK
IF (Alarmes.AlarmeGrave
	//OR NOT Alarmes.AlarmeMedio
	//OR NOT MaquinaLigada
	OR NOT MaquinaModoAuto
	) THEN
	PassoCameraAuto := 1000;
END_IF

CASE PassoCameraAuto OF
	
	//Passo 0 - Inicialização	
	0: PassoCameraAuto := 10;
	   
	//Passo 10 - Condição para Iniciar a Rotina da Camera
	10: IF  (Flag_Robo_Camera) THEN
			Flag_Robo_Camera := FALSE;
			PassoCameraAuto := 20;
		END_IF
		
	//Passo 20 - Set Job
	20: Camera_SetJob := INT_TO_BYTE(Camera_TargetJob[Camera_indexJob]);
		PassoCameraAuto := 21;

	21: Camera_ChangeJob := TRUE;
		TON_CameraChangeJob(IN := TRUE, PT := T#1S);
		IF (TON_CameraChangeJob.Q) THEN
			Camera_ChangeJob := FALSE;
			TON_CameraChangeJob(IN := FALSE);
			PassoCameraAuto := 30;	
		END_IF
		
	//Passo 30 - Disparar Câmera (TRIGGER) 
	30:	Camera_Trigger := TRUE;
		TON_DelayTest1(IN := TRUE, PT := T#1S);
		IF (TON_DelayTest1.Q) THEN
			Camera_Trigger := FALSE;
			TON_DelayTest1(IN := FALSE);
			PassoCameraAuto := 50;	
		END_IF
		//PassoCameraAuto := 40;
		
(*	//Passo 40 - Aguardar Análise da Câmera
	40: //TON_CameraError(IN := TRUE, PT := T#1S);
		IF (Camera_JobCompleted) THEN
			TON_CameraError(IN := FALSE);
			PassoCameraAuto := 50;
		END_IF
		//IF (TON_CameraError.Q) THEN
		//	TON_CameraError(IN := FALSE);
			//Set Flag de Erro
		//	PassoCameraAuto := 50;
		//END_IF
*)		
	//Passo 50 - Sinalizar Resultado da Avaliação
	50: IF (Camera_JobResult) THEN
			PecaAprovada := TRUE;
		ELSE
			PecaAprovada := FALSE;
		END_IF

		PassoCameraAuto := 60;
		
	//Passo 60 - Sinalizar Conclusão da Rotina
	60: Camera_Trigger := FALSE;
		Flag_Camera_Robo := TRUE;
		PassoCameraAuto := 1000;	
	
	//Passo 1000 - Finalização
	1000: PassoCameraAuto := 0;
	
END_CASE

(*========================================================================*)

END_PROGRAM

// ---- POUs/Perifericos/MaquinaSolda.TcPOU
PROGRAM MaquinaSolda
VAR

(*=====================		MÁQUINA DE SOLDA		======================*)	

MaquinaSolda_Receita 		: BYTE;
PassoMaquinaSoldaManual		: INT;
PassoMaquinaSoldaAuto		: INT;
DelayErroMaquinaSoldaManual	: TON;
DelayErroMaquinaSoldaAuto	: TON;
DelayPosicaoCilindro		: TON;

(*========================================================================*)

END_VAR

(*===========		MÁQUINA DE SOLDA - DEFINIÇÃO DE RECEITA		==========*)

	MaquinaSolda_Receita := INT_TO_BYTE(32-1);

	OutMaquinaSolda_Receita_Bit1 := MaquinaSolda_Receita.0;
	OutMaquinaSolda_Receita_Bit2 := MaquinaSolda_Receita.1;
	OutMaquinaSolda_Receita_Bit3 := MaquinaSolda_Receita.2;
	OutMaquinaSolda_Receita_Bit4 := MaquinaSolda_Receita.3;
	OutMaquinaSolda_Receita_Bit5 := MaquinaSolda_Receita.4;
	
(*=================		MÁQUINA DE SOLDA - SAÍDAS		==================*)

	OutMaquinaSolda_BtReset := IhmBt_MaquinaSolda_Reset;

IF(MaquinaModoManual) THEN
	OutMaquinaSolda_BtStart := LigarMaquinaSoldaManual;
ELSIF (MaquinaModoAuto) THEN
	OutMaquinaSolda_BtStart := LigarMaquinaSoldaAuto;
ELSE
	OutMaquinaSolda_BtStart := FALSE;
END_IF

(*=========================		Modo Manual		==========================*)
												
//Condição de Bloqueio da Máquina de Estados - Máquina de Solda Modo Auto
IF (Alarmes.AlarmeGrave
	//OR Alarmes.AlarmeMedio
	//OR Alarmes.AlarmeLeve
	OR NOT MaquinaLigada
	OR NOT MaquinaModoManual
	) THEN
	PassoMaquinaSoldaManual := 1000;
	LigarMaquinaSoldaManual := FALSE;
	DelayErroMaquinaSoldaManual(IN := FALSE);
END_IF

CASE PassoMaquinaSoldaManual OF
	
	//Passo 0 - Inicialização	
	0: PassoMaquinaSoldaManual := 10;
	
	//Passo 10 - Condição para Iniciar a Rotina da Máquina de Solda
	10: IF  (IhmBt_MaquinaSolda_Start) THEN
			PassoMaquinaSoldaManual := 20;
		END_IF

	//Passo 20 - Ligar Máquina de Solda
	20: LigarMaquinaSoldaManual := TRUE;
		DelayErroMaquinaSoldaManual(IN := TRUE, PT := T#4S);
		IF (DelayErroMaquinaSoldaManual.Q) THEN
			DelayErroMaquinaSoldaManual(IN := FALSE);
			LigarMaquinaSoldaManual := FALSE;
			PassoMaquinaSoldaManual := 40;	
		ELSIF (InMaquinaSolda_FK) THEN
			LigarMaquinaSoldaManual := FALSE;
			PassoMaquinaSoldaManual := 30;
		END_IF
		
	//Passo 30 - Fim do Processo de Solda
	30:	DelayErroMaquinaSoldaManual(IN := TRUE, PT := T#4S);
		IF (DelayErroMaquinaSoldaManual.Q) THEN
			DelayErroMaquinaSoldaManual(IN := FALSE);
			LigarMaquinaSoldaManual := FALSE;
			PassoMaquinaSoldaManual := 40;	
		ELSIF (NOT InMaquinaSolda_FK) THEN
			LigarMaquinaSoldaManual := FALSE;
			PassoMaquinaSoldaManual := 40;
		END_IF

	//Passo 40 - Sinalização da Conclusão da Rotina
	40: IhmBt_MaquinaSolda_Start := FALSE;
		PassoMaquinaSoldaManual := 1000;
	
	//Passo 1000 - Finalização
	1000: 	IhmBt_MaquinaSolda_Start := FALSE;
			PassoMaquinaSoldaManual := 0;
	
END_CASE

(*======================		Modo Automático		======================*)

//Condição de Bloqueio da Máquina de Estados - Máquina de Solda Modo Auto
IF (Alarmes.AlarmeGrave
	//OR Alarmes.AlarmeMedio
	//OR Alarmes.AlarmeLeve
	OR NOT MaquinaLigada
	OR NOT MaquinaModoAuto
	) THEN
	PassoMaquinaSoldaAuto := 1000;
	Flag_MaquinaSolda_ServosXY := FALSE;
	LigarMaquinaSoldaAuto := FALSE;
	DelayPosicaoCilindro(IN := FALSE);
END_IF

CASE PassoMaquinaSoldaAuto OF
	
	//Passo 0 - Inicialização	
	0: PassoMaquinaSoldaAuto := 10;
	
	//Passo 10 - Condição para Iniciar a Rotina da Máquina de Solda
	10: IF  (Flag_ServosXY_MaquinaSolda) THEN
			Flag_ServosXY_MaquinaSolda := FALSE;
			PassoMaquinaSoldaAuto := 20;
		END_IF
		
	//Passo 20 - Avançar Cilindro Principal
	20: LigarValvulaY6 := TRUE;
		DelayPosicaoCilindro(IN := TRUE, PT := T#2S);
		IF (DelayPosicaoCilindro.Q) THEN
			DelayPosicaoCilindro(IN := FALSE);
			PassoMaquinaSoldaAuto := 30;
		END_IF
				
	//Passo 30 - Verificar Posição do Cilindro
	30: IF (ReguaPotenciometricaSinal < 29000 AND ReguaPotenciometricaSinal > 28000) THEN
			PassoMaquinaSoldaAuto := 40;
		ELSE
			PassoMaquinaSoldaAuto := 60;
		END_IF

	//Passo 40 - Ligar Máquina de Solda
	40: LigarMaquinaSoldaAuto := TRUE;
		DelayErroMaquinaSoldaAuto(IN := TRUE, PT := T#4S);
		IF (DelayErroMaquinaSoldaAuto.Q) THEN
			DelayErroMaquinaSoldaAuto(IN := FALSE);
			LigarMaquinaSoldaAuto := FALSE;
			PassoMaquinaSoldaAuto := 60;	
		ELSIF (InMaquinaSolda_FK) THEN
			LigarMaquinaSoldaAuto := FALSE;
			PassoMaquinaSoldaAuto := 50;
		END_IF
		
	//Passo 50 - Fim do Processo de Solda
	50:	DelayErroMaquinaSoldaAuto(IN := TRUE, PT := T#2S);
		IF (DelayErroMaquinaSoldaAuto.Q) THEN
			DelayErroMaquinaSoldaAuto(IN := FALSE);
			LigarMaquinaSoldaAuto := FALSE;
			PassoMaquinaSoldaAuto := 60;	
		ELSIF (NOT InMaquinaSolda_FK) THEN
			LigarMaquinaSoldaAuto := FALSE;
			PassoMaquinaSoldaAuto := 50;
		END_IF

	//Passo 60 - Recuar Cilindro Principal
	60: LigarValvulaY6 := FALSE;
		IF (ReguaPotenciometricaSinal > 500 AND ReguaPotenciometricaSinal < 20000) THEN
			PassoMaquinaSoldaAuto := 70;
		END_IF
		
	//Passo 70 - Sinalização da Conclusão da Rotina
	70: Flag_MaquinaSolda_ServosXY := TRUE;
		PassoMaquinaSoldaAuto := 1000;
	
	//Passo 1000 - Finalização
	1000: PassoMaquinaSoldaAuto := 0;
	
END_CASE

(*========================================================================*)

END_PROGRAM

// ---- POUs/IHM.TcPOU
PROGRAM IHM
VAR
		
	SafetyPLCIn 	AT %I*:BYTE;
	SafetyPLCOut 	AT %Q*:BYTE;
	
	sUrlAddressCamera : STRING;

	writeData:FB_WritePersistentData;
	t1:TON;
	bSavePersistent: BOOL;
	
	timer_login	: TON;
	
	Timer_Blink_1hz_1	: TON;
	Timer_Blink_1hz_2	: TON;
	
	b_contador		: BOOL;
	int_contador_10		: INT;
	
	
	PassoBtLigarDesligar	: INT;
	PassoBtReset			: INT;
	PassoMaquina			: INT;
	
END_VAR

(*=====================		STATUS DA MÁQUINA		======================*)

//Máquina em Alarme
IF (Alarmes.AlarmeGrave
	)THEN	
	MaquinaAlarme := TRUE;
ELSE
	MaquinaAlarme := FALSE;
END_IF	

(*=====================		LÓGICA DOS BOTÕES		======================*)

(*=====================		LIGAR E DESLIGAR		======================*)

//Condição de Bloqueio da Máquina de Estados - Botões Ligar e Desligar
IF (Alarmes.AlarmeGrave
	//OR Alarmes.AlarmeMedio
	//OR Alarmes.AlarmeLeve
	OR MaquinaModoManual
	) THEN
	PassoBtLigarDesligar := 1000;
	IhmBt_Desligar := TRUE;
	IhmBt_Ligar := FALSE;
	Flag_CondicoesIniciais := TRUE;
END_IF

// Máquina de Estados - Botões Ligar e Desligar
CASE PassoBtLigarDesligar OF

	//Passo 0 - Inicialização
	0: PassoBtLigarDesligar := 10;
	
	//Passo 10 - Botão Ligar
	10: IF IhmBt_Ligar THEN
			MaquinaLigada := TRUE;
			PassoBtLigarDesligar := 20;
			IhmBt_Ligar := TRUE;
			IhmBt_Desligar := FALSE;
		ELSIF NOT IhmBt_Ligar THEN
			IhmBt_Desligar := TRUE;
		END_IF
	
	//Passo 20 - Botão Desligar
	20: IF IhmBt_Desligar THEN
			MaquinaLigada := FALSE;
			PassoBtLigarDesligar := 1000;
			IhmBt_Ligar := FALSE;
			IhmBt_Desligar := TRUE;
		ELSIF NOT IhmBt_Ligar THEN
			IhmBt_Ligar := TRUE;
		END_IF
	
	//Passo 1000 - Finalização
	1000: PassoBtLigarDesligar := 0;

END_CASE

(*==========================		RESET		==========================*)

IF (InSolicitaReset OR IhmBt_Reset) THEN
	Reset := TRUE;
ELSE
	Reset := FALSE;
END_IF

(*=====================		MODO MANUAL / AUTO		======================*)

IF IhmBt_ManualAuto THEN
	IhmBt_ManualAuto_Text := 'MANUAL';
	IhmBt_ManualAuto_Color := TRUE;
	MaquinaModoManual := TRUE;
	MaquinaModoAuto := FALSE;
ELSE
	IhmBt_ManualAuto_Text := 'AUTO';
	IhmBt_ManualAuto_Color := FALSE;
	MaquinaModoManual := FALSE;
	MaquinaModoAuto := TRUE;
END_IF

(*========================================================================*)


(*========================================================================*)

//				Hora do Sistema					\\
	FB_HoraAtual (START := TRUE, TIMESTR => tempo);
	FB_HoraAtual (START := FALSE);
	TempoAtual := SYSTEMTIME_TO_DT (tempo);

t1(IN:= NOT t1.Q, PT:=T#1M);	
writeData(
	NETID:='' , 
	PORT:=851 , 
	START:= t1.Q OR bSavePersistent, 
	TMOUT:= T#10S, 
	MODE:= , 
	BUSY=> , 
	ERR=> ,  
	ERRID=> );	
	
	UserGroupName 	:= WSTRING_TO_STRING (visuelems.CurrentUserGroupName);
	UserGroupId		:= (visuelems.CurrentUserGroupId);

IF UserGroupId = 1 THEN
	UserName := WSTRING_TO_STRING(VisuElems.CurrentUserName);
	timer_login (in := FALSE);
	
ELSIF UserGroupId = 0 THEN
	timer_login (in := TRUE, pt := T#1S);	
	IF timer_login.Q THEN
		UserName := '';
		b_editar_receita := FALSE;
	END_IF
END_IF

(*///////////////////////////////			BLINK 0.25 HZ		\\\\\\\\\\\\\\\\\\\\\\\\\\\\\\\\\\\\\\\
IF IhmBt_Ligar THEN
	Timer_Blink_1hz_1 (IN := TRUE, PT := T#2S);	
END_IF

IF Timer_Blink_1hz_1.Q THEN
	Blink_1hz := TRUE;
	Timer_Blink_1hz_2 (IN := TRUE, PT := T#2S);
	IF Timer_Blink_1hz_2.Q THEN
		Blink_1hz := FALSE;
		Timer_Blink_1hz_1 (IN := FALSE);
		Timer_Blink_1hz_2 (IN := FALSE);
	END_IF
END_IF

	I2 := Blink_1hz;
	
	IF NOT b_contador AND Blink_1hz THEN
		b_contador := TRUE;
		Contador_Total := Contador_Total + 1;
		Contador_Pecas_Boas := Contador_Pecas_Boas + 1;
		int_contador_10 := int_contador_10 + 1;
	END_IF
	IF NOT Blink_1hz THEN
		b_contador := FALSE;
	END_IF
	
	IF int_contador_10 = 10 THEN
		int_contador_10 := 0;
		Contador_Pecas_Boas := Contador_Pecas_Boas - 1;
		Contador_Refugo := Contador_Refugo + 1;
	END_IF
*)	
	IF BT_ihm_zerar_contador THEN
		BT_ihm_zerar_contador := FALSE;
		Contador_Total := 0;
		Contador_PecasAprovadas := 0;
		Contador_PecasReprovadas := 0;
	END_IF

END_PROGRAM

// ---- POUs/Sinalizadores.TcPOU
PROGRAM Sinalizadores
VAR
END_VAR

(*=================		SINALIZADORES LUMINOSOS		======================*)	

//Comando Ligado
IF (TRUE) THEN
	OutSinalizadorComandoLigado := TRUE;
ELSE
	OutSinalizadorComandoLigado := FALSE;
END_IF

//Botoeira HS1
IF (TRUE) THEN
	OutSinalizadorBotoeiraHS1 := TRUE;
ELSE
	OutSinalizadorBotoeiraHS1 := FALSE;
END_IF

//Botoeira HS2
IF (TRUE) THEN
	OutSinalizadorBotoeiraHS2 := TRUE;
ELSE
	OutSinalizadorBotoeiraHS2 := FALSE;
END_IF

(*========================================================================*)

END_PROGRAM

// ---- POUs/Perifericos/SafetyPLC.TcPOU
PROGRAM SafetyPLC
VAR

(*=========================		SAFETY PLC		==========================*)	



(*========================================================================*)

END_VAR

(*=========================		SAFETY PLC		==========================*)



(*========================================================================*)

END_PROGRAM

// ---- GlobalTextList.TcGTLO
TEXTLIST GlobalTextList
  2346 = ' STATUS %s '
  2796 = ' STATUS %s "'
  2282 = '%'
  582 = '% Cilindro'
  2657 = '% Válvula Proporcional'
  2893 = '%.2F'
  4433 = '%.2f %'
  1907 = '%.2f mm'
  4611 = '%.2f mm/s'
  742 = '%.2f s'
  2952 = '%1.2f %'
  1098 = '%1.2f mm/s'
  1576 = '%1.2f s'
  50 = '%d'
  2982 = '%d %'
  3579 = '%d 5'
  1770 = '%d Hz'
  1788 = '%d kgf'
  1253 = '%d kgfm'
  4006 = '%d m'
  2537 = '%d mm'
  3937 = '%d mm/s'
  150 = '%d Peças'
  1343 = '%d RPM'
  1397 = '%d s'
  1299 = '%s'
  2396 = '%s '
  1289 = '%s mm'
  2879 = '%s s'
  798 = '%t[dd/MM/yyyy]'
  720 = '%t[HH:mm:ss]'
  219 = '(mm)'
  3796 = '(Sensor Fim de Curso)'
  3320 = '(Válvula Y1)'
  2536 = '1 mm/s'
  2851 = '1° Ponto - (X,Y)'
  573 = '1° Ponto - X'
  2310 = '1° Ponto - Y'
  441 = '2 - Entrada Digital 2'
  1114 = '2 - Entrada Digital 50'
  182 = '2° Ponto - (X,Y)'
  599 = '2° Ponto - X'
  1505 = '2° Ponto - Y'
  1844 = '3° Ponto - (X,Y)'
  622 = '3° Ponto - X'
  1502 = '3° Ponto - Y'
  132 = '49 - Entrada Digital 1'
  2798 = '4° Ponto - (X,Y)'
  810 = '4° Ponto - X'
  283 = '50 - Entrada Digital 2'
  1649 = '5° Ponto - (X,Y)'
  2974 = '5° Ponto - X'
  1148 = '6° Ponto - X'
  2872 = 'Abertura da Porta da Câmera'
  1259 = 'Abertura da Porta da Esteira'
  288 = 'Abertura da Porta da Máquina de Solda / Robô'
  521 = 'Abertura da Porta do Painel Principal'
  2773 = 'Abertura da Porta Frontal Inferior'
  2479 = 'Abertura da Porta Lateral Esquerda - Folha Direita'
  636 = 'Abertura da Porta Lateral Esquerda - Folha Esquerda'
  2720 = 'Abrir'
  740 = 'Admin'
  550 = 'Administrador: %s'
  597 = 'Ajustes - Câmera'
  2048 = 'Ajustes - Inversores'
  3983 = 'Ajustes - Servos'
  366 = 'ALARMES'
  3308 = 'ALARMES - Configurações'
  1463 = 'ALARMES - PAINEL PNEUMÁTICO'
  793 = 'ALARMES DE ABERTURA DE PORTAS'
  188 = 'ALARMES DE EMERGÊNCIA'
  908 = 'AO1 - Saida Analogica 1'
  838 = 'AO1 - Saida Analogica 2'
  524 = 'AO1 - Saida Analogica 3'
  1706 = 'AO1 - Saida Analogica 4'
  2466 = 'Bloco de Válvulas'
  3692 = 'Botão de Emergência da Porta M/áq. Solda'
  2330 = 'Botão de Emergência da Porta Maq. Solda'
  4548 = 'Botão de Emergência da Porta Máq. Solda'
  529 = 'Botão de Emergência do Chiller'
  2903 = 'Botão de Emergência do Robô'
  4578 = 'Botão de Emergência Frontal'
  4374 = 'CAIXA'
  4134 = 'CALIBRAR'
  338 = 'Calibrar Avanço'
  819 = 'Calibrar Porca'
  4743 = 'Calibrar Recuo'
  1497 = 'Camera Sick Inspector'
  1826 = 'CANCELA'
  1667 = 'CANCELAR'
  2511 = 'CHANGE JOG'
  1973 = 'COMANDOS'
  2850 = 'COND. INICIAIS'
  816 = 'Conexão Ethernet/IP'
  1413 = 'Controle Manual:'
  1838 = 'Create Recipe'
  2650 = 'CÂMERA'
  3559 = 'Delay (ERROR):'
  4227 = 'Delay (Parada)'
  1168 = 'DELETAR'
  2254 = 'delete'
  51 = 'DESCARTE'
  3936 = 'Deslocar 1 Posição'
  834 = 'dgdfg'
  299 = 'Dispositivos Safety'
  2227 = 'Editar'
  2382 = 'EDITAR'
  2487 = 'Editar Receita'
  385 = 'EL1809 - Cartão 16 Entradas Digitais'
  2710 = 'ELEMENTOS PNEUMÁTICOS'
  1312 = 'Excluir'
  358 = 'Excluir Receita'
  1921 = 'Excluir Receita  Selecionada'
  1853 = 'Excluir Receita Selecionada'
  1280 = 'Excluir ReceitaSelecionada'
  857 = 'Executando Job (Job ID):'
  828 = 'EXECUTAR'
  158 = 'Executar Receita'
  892 = 'F01'
  3241 = 'F02'
  2098 = 'F03'
  4267 = 'F04'
  2725 = 'F05'
  3970 = 'FERRAMENTA'
  1076 = 'FIM DE CURSO'
  436 = 'Foto'
  2367 = 'Frequência (Esteira):'
  803 = 'Frequência (Mesa):'
  340 = 'FX3 - XTIO84002 - 8 entradas e 4 Saídas'
  379 = 'Garra do Robô'
  228 = 'HOME'
  540 = 'I1 - Entrada Digital 1'
  545 = 'I1 - Entrada Digital 1 - Botão de Emergencia '
  1767 = 'I1 - Entrada Digital 1 - Sensor Atuador Rec'
  603 = 'I1 - Entrada Digital 10'
  913 = 'I1 - Entrada Digital 11'
  997 = 'I1 - Entrada Digital 12'
  635 = 'I1 - Entrada Digital 13'
  26 = 'I1 - Entrada Digital 14'
  113 = 'I1 - Entrada Digital 15'
  734 = 'I1 - Entrada Digital 16'
  203 = 'I1 - Entrada Digital 17'
  531 = 'I1 - Entrada Digital 2'
  668 = 'I1 - Entrada Digital 3'
  528 = 'I1 - Entrada Digital 31'
  310 = 'I1 - Entrada Digital 33'
  480 = 'I1 - Entrada Digital 4'
  869 = 'I1 - Entrada Digital 49'
  383 = 'I1 - Entrada Digital 5'
  858 = 'I1 - Entrada Digital 6'
  789 = 'I1 - Entrada Digital 7'
  925 = 'I1 - Entrada Digital 8'
  578 = 'I1 - Entrada Digital 9'
  650 = 'I1 - Entrada Rapida 1'
  1222 = 'I1 - Saida Digital 1'
  753 = 'I1-I2 - Botão de Emergência'
  2080 = 'I1-I2 - Cortina de Luz'
  999 = 'I1-I2 - Sensor Porta'
  905 = 'I10 - Entrada Digital 10'
  160 = 'I10 - Entrada Digital 26'
  506 = 'I10 - Entrada Digital 42'
  171 = 'I10 - Entrada Digital 58'
  281 = 'I10 - Saida Digital 10'
  505 = 'I11 - Entrada Digital 11'
  631 = 'I11 - Entrada Digital 27'
  374 = 'I11 - Entrada Digital 43'
  69 = 'I11 - Entrada Digital 59'
  396 = 'I11 - Saida Digital 11'
  481 = 'I12 - Entrada Digital 12'
  5 = 'I12 - Entrada Digital 28'
  558 = 'I12 - Entrada Digital 44'
  408 = 'I12 - Entrada Digital 60'
  895 = 'I12 - Saida Digital 12'
  885 = 'I13 - Entrada Digital 13'
  710 = 'I13 - Entrada Digital 29'
  911 = 'I13 - Entrada Digital 45'
  177 = 'I13 - Entrada Digital 61'
  689 = 'I13 - Saida Digital 13'
  36 = 'I14 - Entrada Digital 14'
  735 = 'I14 - Entrada Digital 30'
  81 = 'I14 - Entrada Digital 46'
  926 = 'I14 - Entrada Digital 62'
  560 = 'I14 - Saida Digital 14'
  99 = 'I15 - Entrada Digital 15'
  463 = 'I15 - Entrada Digital 31'
  713 = 'I15 - Entrada Digital 47'
  921 = 'I15 - Entrada Digital 63'
  1398 = 'I15 - Saida Digital 15'
  361 = 'I16 - Entrada Digital 16'
  115 = 'I16 - Entrada Digital 32'
  693 = 'I16 - Entrada Digital 48'
  180 = 'I16 - Entrada Digital 64'
  418 = 'I16 - Saida Digital 16'
  372 = 'I17 - Entrada Digital 1'
  701 = 'I18 - Entrada Digital 2'
  287 = 'I19 - Entrada Digital 3'
  995 = 'I2 - Entrada Digital 18'
  730 = 'I2 - Entrada Digital 2'
  1430 = 'I2 - Entrada Digital 31'
  63 = 'I2 - Entrada Digital 34'
  339 = 'I2 - Entrada Digital 50'
  1472 = 'I2 - Entrada Rapida 2'
  470 = 'I2 - Saida Digital 2'
  804 = 'I20 - Entrada Digital 4'
  258 = 'I21 - Entrada Digital 5'
  269 = 'I22 - Entrada Digital 6'
  443 = 'I23 - Entrada Digital 7'
  448 = 'I24 - Entrada Digital 8'
  476 = 'I25 - Entrada Digital 9'
  373 = 'I26 - Entrada Digital 10'
  353 = 'I27 - Entrada Digital 11'
  821 = 'I28 - Entrada Digital 12'
  571 = 'I29 - Entrada Digital 13'
  184 = 'I3 - Entrada Digital 19'
  971 = 'I3 - Entrada Digital 3'
  538 = 'I3 - Entrada Digital 35'
  886 = 'I3 - Entrada Digital 51'
  935 = 'I3 - Saida Digital 3'
  163 = 'I3-I4 - Botão de Emergência'
  2387 = 'I3-I4 - Sensor Porta'
  771 = 'I30 - Entrada Digital 14'
  584 = 'I31 - Entrada Digital 15'
  31 = 'I32 - Entrada Digital 16'
  806 = 'I33 - Entrada Digital 1'
  811 = 'I34 - Entrada Digital 2'
  833 = 'I35 - Entrada Digital 3'
  645 = 'I36 - Entrada Digital 4'
  256 = 'I37 - Entrada Digital 5'
  382 = 'I38 - Entrada Digital 6'
  799 = 'I39 - Entrada Digital 7'
  390 = 'I4 - Entrada Digital 20'
  298 = 'I4 - Entrada Digital 36'
  437 = 'I4 - Entrada Digital 4'
  739 = 'I4 - Entrada Digital 52'
  149 = 'I4 - Saida Digital 4'
  572 = 'I40 - Entrada Digital 8'
  918 = 'I41 - Entrada Digital 9'
  654 = 'I42 - Entrada Digital 10'
  28 = 'I43 - Entrada Digital 11'
  74 = 'I44 - Entrada Digital 12'
  633 = 'I45 - Entrada Digital 13'
  34 = 'I46 - Entrada Digital 14'
  916 = 'I47 - Entrada Digital 15'
  49 = 'I48 - Entrada Digital 16'
  7 = 'I49 - Entrada Digital 1'
  934 = 'I5 - Entrada Digital 21'
  413 = 'I5 - Entrada Digital 37'
  318 = 'I5 - Entrada Digital 5'
  342 = 'I5 - Entrada Digital 53'
  286 = 'I5 - Saida Digital 5'
  755 = 'I51 - Entrada Digital 3'
  902 = 'I52 - Entrada Digital 4'
  321 = 'I53 - Entrada Digital 5'
  144 = 'I54 - Entrada Digital 6'
  945 = 'I6 - Entrada Digital 22'
  83 = 'I6 - Entrada Digital 38'
  225 = 'I6 - Entrada Digital 54'
  238 = 'I6 - Entrada Digital 6'
  688 = 'I6 - Entrada Digital54'
  87 = 'I6 - Saida Digital 6'
  402 = 'I7 - Entrada Digital 23'
  507 = 'I7 - Entrada Digital 39'
  823 = 'I7 - Entrada Digital 55'
  535 = 'I7 - Entrada Digital 7'
  344 = 'I7 - Saida Digital 7'
  162 = 'I8 - Entrada Digital 24'
  539 = 'I8 - Entrada Digital 40'
  859 = 'I8 - Entrada Digital 56'
  773 = 'I8 - Entrada Digital 8'
  1097 = 'I8 - Saida Digital 8'
  170 = 'I9 - Entrada Digital 25'
  812 = 'I9 - Entrada Digital 41'
  1133 = 'I9 - Entrada Digital 57'
  485 = 'I9 - Entrada Digital 9'
  1096 = 'I9 - Saida Digital 9'
  5145 = 'ID'
  2239 = 'ID: %d'
  4583 = 'ID: %s'
  3757 = 'INICIO CURSO'
  1135 = 'INICIO DE CURSO'
  2585 = 'Inv. Esteira'
  2998 = 'Inv. Mesa'
  1439 = 'Inversor Esteira'
  1539 = 'Inversor Mesa'
  4459 = 'INÍCIO DE CURSO'
  127 = 'Job Completed:'
  3080 = 'Job ID: %s'
  2980 = 'Job Result:'
  1782 = 'JOG'
  1089 = 'kjhfg'
  2787 = 'Liga/Desliga'
  1768 = 'Load from file'
  2469 = 'LOGIN'
  1255 = 'login'
  1329 = 'Login'
  14 = 'logout'
  1939 = 'Logout'
  557 = 'MANUAL'
  808 = 'manutenção'
  2820 = 'MANUTENÇÃO'
  2550 = 'MARCELO'
  1956 = 'mm'
  254 = 'MODO AUTOMÁTICO'
  4429 = 'MODO: '
  4753 = 'MODO: %s'
  4355 = 'Monitaramento'
  1855 = 'Monitoramento'
  2574 = 'MOTORES'
  2424 = 'MOTORES E CÂMERA'
  1318 = 'MOV. MANUAIS'
  2535 = 'MOVIMENTOS MANUAIS'
  1082 = 'mudar senha'
  928 = 'Mudar senha'
  1268 = 'Máquina de Solda'
  2708 = 'MÁQUINA DE SOLDA'
  4465 = 'No.'
  2481 = 'Nome da Receita: %s'
  1532 = 'Nome: %s'
  809 = 'None'
  936 = 'Nova Receita'
  2159 = 'N° Peças por Caixa'
  29 = 'Número de Fotos'
  2956 = 'Número de Pontos'
  2113 = 'Operator'
  4168 = 'OPERAÇÃO'
  604 = 'Operação'
  1361 = 'P01 - (X,Y)'
  2292 = 'P02 - (X,Y)'
  826 = 'P03 - (X,Y)'
  3609 = 'P04 - (X,Y)'
  3644 = 'P05 - (X,Y)'
  3275 = 'P06 - (X,Y'
  3037 = 'P06 - (X,Y)'
  1504 = 'P07 - (X,Y)'
  1202 = 'P08 - (X,Y'
  1084 = 'P08 - (X,Y)'
  1549 = 'P09 - (X,Y)'
  746 = 'P10 - (X,Y)'
  1319 = 'P11 - (X,Y)'
  116 = 'P12 - (X,Y)'
  738 = 'P13 - (X,Y)'
  3363 = 'P14 - (X,Y)'
  2712 = 'P15 - (X,Y)'
  3015 = 'P16 - (X,Y)'
  906 = 'P17 - (X,Y)'
  322 = 'P18 - (X,Y)'
  2901 = 'P19 - (X,Y)'
  1216 = 'P20 - (X,Y)'
  570 = 'PAUSE'
  25 = 'Pega do Robo - (X,Y'
  933 = 'Pega do Robo - (X,Y, Z)'
  360 = 'Pega do Robo - (X,Y,Z)'
  2894 = 'Pega do Robo - (X,YZ)'
  2422 = 'Pega do Robo - X'
  85 = 'Pega do Robo - Y'
  835 = 'PEGA PEÇA'
  3889 = 'Pos. Manual'
  1324 = 'POS. ZERO'
  3752 = 'Posição'
  3255 = 'Posições Fixas'
  1402 = 'POWER ON'
  2624 = 'Pressostato Geral (Digital)'
  3890 = 'PRESSÃO NORMAL'
  89 = 'PRODUÇÃO'
  752 = 'PROGRAMA '
  1650 = 'PROGRAMA "%s "'
  3334 = 'PROGRAMA "%s"'
  1522 = 'PROGRAMA: "%s "'
  1748 = 'PROGRAMA: "%S"'
  996 = 'PROGRAMA: "%s"'
  907 = 'Q1 - Saida Digital 1'
  846 = 'Q1 - Saida Digital 17'
  391 = 'Q1 - Saida Digital 33'
  1238 = 'Q1 - Saida Digital 49'
  665 = 'Q1-Q2 - Botão de Emergência'
  400 = 'Q1-Q2 - Motor '
  1039 = 'Q1-Q2 - Robo Yaskawa GP7'
  239 = 'Q1-Q2 - Servo 1'
  552 = 'Q10 - Saida Digital 10'
  1257 = 'Q10 - Saida Digital 26'
  839 = 'Q10 - Saida Digital 42'
  304 = 'Q10 - Saida Digital 58'
  519 = 'Q11 - Saida Digital 11'
  375 = 'Q11 - Saida Digital 27'
  1059 = 'Q11 - Saida Digital 43'
  61 = 'Q11 - Saida Digital 59'
  1491 = 'Q12 - Saida Digital 12'
  111 = 'Q12 - Saida Digital 28'
  1499 = 'Q12 - Saida Digital 44'
  527 = 'Q12 - Saida Digital 60'
  467 = 'Q13 - Saida Digital 13'
  1058 = 'Q13 - Saida Digital 29'
  695 = 'Q13 - Saida Digital 45'
  736 = 'Q13 - Saida Digital 61'
  121 = 'Q14 - Saida Digital 14'
  1488 = 'Q14 - Saida Digital 30'
  877 = 'Q14 - Saida Digital 46'
  791 = 'Q14 - Saida Digital 62'
  1567 = 'Q15 - Saida Digital 15'
  369 = 'Q15 - Saida Digital 31'
  1242 = 'Q15 - Saida Digital 47'
  319 = 'Q15 - Saida Digital 63'
  1359 = 'Q16 - Saida Digital 16'
  682 = 'Q16 - Saida Digital 32'
  1401 = 'Q16 - Saida Digital 48'
  376 = 'Q16 - Saida Digital 64'
  1212 = 'Q2 - Saida Digital 18'
  870 = 'Q2 - Saida Digital 2'
  438 = 'Q2 - Saida Digital 34'
  556 = 'Q2 - Saida Digital 50'
  790 = 'Q3 - Saida Digital 19'
  1444 = 'Q3 - Saida Digital 3'
  722 = 'Q3 - Saida Digital 35'
  1060 = 'Q3 - Saida Digital 51'
  2293 = 'Q3-Q4 - Botão de Emergência'
  1544 = 'Q3-Q4 - Motor'
  1458 = 'Q3-Q4 - Reserva'
  1526 = 'Q3-Q4 - Robo Yaskawa GP7'
  1048 = 'Q3-Q4 - Servo 2'
  837 = 'Q4 - Saida Digital 20'
  246 = 'Q4 - Saida Digital 36'
  297 = 'Q4 - Saida Digital 4'
  1254 = 'Q4 - Saida Digital 52'
  982 = 'Q5 - Saida Digital 21'
  1712 = 'Q5 - Saida Digital 37'
  493 = 'Q5 - Saida Digital 5'
  1821 = 'Q5 - Saida Digital 53'
  187 = 'Q6 - Saida Digital 22'
  1438 = 'Q6 - Saida Digital 38'
  1586 = 'Q6 - Saida Digital 54'
  293 = 'Q6 - Saida Digital 6'
  1226 = 'Q7 - Saida Digital 23'
  516 = 'Q7 - Saida Digital 39'
  549 = 'Q7 - Saida Digital 55'
  883 = 'Q7 - Saida Digital 7'
  1151 = 'Q8 - Saida Digital 24'
  193 = 'Q8 - Saida Digital 40'
  1918 = 'Q8 - Saida Digital 56'
  847 = 'Q8 - Saida Digital 8'
  963 = 'Q9 - Saida Digital 25'
  1867 = 'Q9 - Saida Digital 41'
  215 = 'Q9 - Saida Digital 57'
  97 = 'Q9 - Saida Digital 9'
  1119 = 'Read'
  1874 = 'receita'
  2877 = 'RECEITAS'
  1575 = 'REF. AUTO'
  1914 = 'REFERENCIAR'
  3213 = 'Reserva'
  341 = 'RESERVA'
  2144 = 'RESET'
  1309 = 'Revolução'
  311 = 'Robo Yaskawa GP7'
  4381 = 'ROBÔ'
  3731 = 'RÉGUA POTENCIOMÉTRICA'
  337 = 's s'
  240 = 'Safety Sick Flexi Soft'
  2485 = 'Salvar'
  2968 = 'SALVAR'
  1252 = 'save'
  2494 = 'Selecionar Job (Job ID):'
  4791 = 'Selecionar Job:'
  1271 = 'Selecionar Receita'
  3057 = 'Sensor Indutivo Válvula de Segurança V7'
  1331 = 'Sensor Indutivo Válvula de Segurança V8'
  488 = 'Service'
  147 = 'SERVO ON'
  663 = 'Servo X'
  1758 = 'Servo Y'
  88 = 'SETUP FERR.'
  2573 = 'SETUP FERRAMENTA'
  2925 = 'Solda'
  2161 = 'START'
  1635 = 'Status Câmera'
  1266 = 'STOP'
  2841 = 'Tela de Manutenção'
  3071 = 'Tela de Rece'
  2618 = 'TELA DE RECEITA'
  1837 = 'Tela de Receitas'
  30 = 'TELA MANUTENÇÃO'
  1963 = 'TELA MENU'
  1042 = 'TELA MOVIMENTOS MANUAIS'
  2878 = 'TELA PRINCIPAL'
  1776 = 'TELA PRODUÇÃO'
  634 = 'TELA RECEITA'
  2326 = 'Tempo (Torque Máximo):'
  2347 = 'Tempo Ciclo Atual'
  2652 = 'Tempo Ciclo Atual: %d seg.'
  1794 = 'TEMPOS'
  876 = 'Term 2 - EL1809 - 16 Entradas Digitais'
  326 = 'Term 3 - EL1809 - 16 Entradas Digitais'
  745 = 'Term 4 - EL1809 - 16 Entradas Digitais'
  836 = 'Term 5 - EL1809 - 16 Entradas Digitais'
  235 = 'Term 6 - EL2809 - 16 Saídas Digitais'
  1142 = 'Term 7 - EL2809 - 16 Saídas Digitais'
  937 = 'Term 8 - EL2809 - 16 Saídas Digitais'
  359 = 'Term 9 - EL1252 - 2 Entradas Rápidas'
  1021 = 'Term 9 - EL2809 - 16 Saídas Digitais'
  1647 = 'Term 9 - EL3064 - 4 Entradas Analógicas'
  1315 = 'Term 9 - EL4004 - 4 Saídas Analógicas'
  2044 = 'TESTE'
  3256 = 'Tolerância (%):'
  17 = 'Torque Máximo:'
  1330 = 'Torque:'
  2934 = 'Total de Peças Aprovadas'
  2195 = 'Total de Peças BOAS'
  2294 = 'Total de Peças Produzida'
  435 = 'Total de Peças Produzidas'
  1862 = 'Total de Peças REFUGO'
  2595 = 'Total de Peças Reprovadas'
  1409 = 'TRIGGER'
  1897 = 'Usuário: %s'
  1043 = 'Velocidade'
  363 = 'Velocidade (Auto)'
  2911 = 'Velocidade (Auto):'
  3254 = 'Velocidade (Manual)'
  1842 = 'Velocidade (Manual):'
  574 = 'Velocidade Manual'
  2412 = 'Velocidade:'
  1403 = 'Válvula Proporcial'
  2569 = 'Válvula Proporcional'
  1104 = 'Válvula Y1'
  3504 = 'Válvula Y10'
  241 = 'Válvula Y11'
  186 = 'Válvula Y12'
  875 = 'Válvula Y2'
  202 = 'Válvula Y3'
  2070 = 'Válvula Y4'
  1218 = 'Válvula Y5'
  3239 = 'Válvula Y6'
  2771 = 'Válvula Y7'
  3632 = 'Válvula Y8'
  1152 = 'Válvula Y9'
  1898 = 'Válvulas de Segurança'
  200 = 'VÁLVULAS DE SEGURANÇA'
  2889 = 'wewerw'
  605 = 'write'
  3482 = 'x1'
  4174 = 'x10'
  1179 = 'x100'
  616 = 'XTIO[1] - 8 entradas e 4 Saídas'
  100 = 'XTIO[2] - 8 entradas e 4 Saídas'
  114 = 'XTIO[3] - 8 entradas e 4 Saídas'
  92 = 'Zerar Contador'
  2498 = 'ZERAR CONTADORES'
  1733 = '± %1.2f %'
  5146 = '± %d %'
  4942 = '± %d Hz'
END_TEXTLIST

// ---- VISUs/Lista_PontosSolda.TcVIS
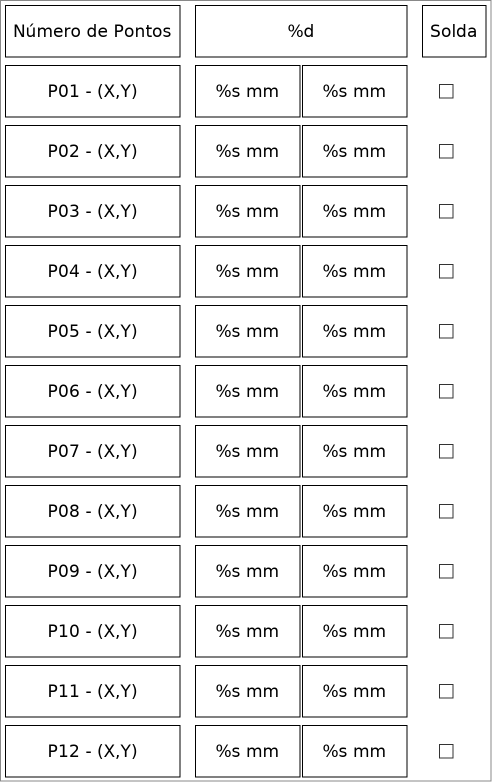
VISUALIZATION Lista_PontosSolda  // 492x782
    Rectangle (5,5 175x52), "Número de Pontos"
    Rectangle (195,5 212x52), "%d", text variable: Recipe_Pontos_Solda_Select, input disabled if: Not b_editar_receita and Not b_criar_receita
        OnMouseClick: write the text variable via Default, min 0, max 5
    Rectangle (5,65 175x52), "P01 - (X,Y)", invisible if: Recipe_Pontos_Solda_Select<1
    Rectangle (195,65 105x52), "%s mm", text variable: Recipe_P_X01_Solda_Select, invisible if: Recipe_Pontos_Solda_Select<1, input disabled if: Not b_editar_receita and Not b_criar_receita
        OnMouseClick: write the text variable via Default, min 0, max 300
    Rectangle (5,125 175x52), "P02 - (X,Y)", invisible if: Recipe_Pontos_Solda_Select<2
    Rectangle (195,125 105x52), "%s mm", text variable: Recipe_P_X02_Solda_Select, invisible if: Recipe_Pontos_Solda_Select<2, input disabled if: Not b_editar_receita and Not b_criar_receita
        OnMouseClick: write the text variable via Default, min 0, max 300
    Rectangle (5,185 175x52), "P03 - (X,Y)", invisible if: Recipe_Pontos_Solda_Select<3
    Rectangle (195,185 105x52), "%s mm", text variable: Recipe_P_X03_Solda_Select, invisible if: Recipe_Pontos_Solda_Select<3, input disabled if: Not b_editar_receita and Not b_criar_receita
        OnMouseClick: write the text variable via Default, min 0, max 300
    Rectangle (5,245 175x52), "P04 - (X,Y)", invisible if: Recipe_Pontos_Solda_Select<4
    Rectangle (195,245 105x52), "%s mm", text variable: Recipe_P_X04_Solda_Select, invisible if: Recipe_Pontos_Solda_Select<4, input disabled if: Not b_editar_receita and Not b_criar_receita
        OnMouseClick: write the text variable via Default, min 0, max 300
    Rectangle (5,305 175x52), "P05 - (X,Y)", invisible if: Recipe_Pontos_Solda_Select<5
    Rectangle (195,305 105x52), "%s mm", text variable: Recipe_P_X05_Solda_Select, invisible if: Recipe_Pontos_Solda_Select<5, input disabled if: Not b_editar_receita and Not b_criar_receita
        OnMouseClick: write the text variable via Default, min 0, max 300
    Rectangle (302,65 105x52), "%s mm", text variable: Recipe_P_Y01_Solda_Select, invisible if: Recipe_Pontos_Solda_Select<1, input disabled if: Not b_editar_receita and Not b_criar_receita
        OnMouseClick: write the text variable via Default, min 0, max 300
    Rectangle (302,125 105x52), "%s mm", text variable: Recipe_P_Y02_Solda_Select, invisible if: Recipe_Pontos_Solda_Select<2, input disabled if: Not b_editar_receita and Not b_criar_receita
        OnMouseClick: write the text variable via Default, min 0, max 300
    Rectangle (302,185 105x52), "%s mm", text variable: Recipe_P_Y03_Solda_Select, invisible if: Recipe_Pontos_Solda_Select<3, input disabled if: Not b_editar_receita and Not b_criar_receita
        OnMouseClick: write the text variable via Default, min 0, max 300
    Rectangle (302,245 105x52), "%s mm", text variable: Recipe_P_Y04_Solda_Select, invisible if: Recipe_Pontos_Solda_Select<4, input disabled if: Not b_editar_receita and Not b_criar_receita
        OnMouseClick: write the text variable via Default, min 0, max 300
    Rectangle (302,305 105x52), "%s mm", text variable: Recipe_P_Y05_Solda_Select, invisible if: Recipe_Pontos_Solda_Select<5, input disabled if: Not b_editar_receita and Not b_criar_receita
        OnMouseClick: write the text variable via Default, min 0, max 300
    Rectangle (422,5 64x52), "Solda"
    Checkbox (437,71 40x40), variable: Recipe_P01_Solda_Select, invisible if: Recipe_Pontos_Solda_Select<1, input disabled if: Not b_editar_receita and Not b_criar_receita
    Checkbox (437,131 40x40), variable: Recipe_P02_Solda_Select, invisible if: Recipe_Pontos_Solda_Select<2, input disabled if: Not b_editar_receita and Not b_criar_receita
    Checkbox (437,191 40x40), variable: Recipe_P03_Solda_Select, invisible if: Recipe_Pontos_Solda_Select<3, input disabled if: Not b_editar_receita and Not b_criar_receita
    Checkbox (437,251 40x40), variable: Recipe_P04_Solda_Select, invisible if: Recipe_Pontos_Solda_Select<4, input disabled if: Not b_editar_receita and Not b_criar_receita
    Checkbox (437,311 40x40), variable: Recipe_P05_Solda_Select, invisible if: Recipe_Pontos_Solda_Select<5, input disabled if: Not b_editar_receita and Not b_criar_receita
    Rectangle (5,365 175x52), "P06 - (X,Y)", invisible if: Recipe_Pontos_Solda_Select<6
    Rectangle (195,365 105x52), "%s mm", text variable: Recipe_P_X06_Solda_Select, invisible if: Recipe_Pontos_Solda_Select<6, input disabled if: Not b_editar_receita and Not b_criar_receita
        OnMouseClick: write the text variable via Default, min 0, max 300
    Rectangle (5,425 175x52), "P07 - (X,Y)", invisible if: Recipe_Pontos_Solda_Select<7
    Rectangle (195,425 105x52), "%s mm", text variable: Recipe_P_X07_Solda_Select, invisible if: Recipe_Pontos_Solda_Select<7, input disabled if: Not b_editar_receita and Not b_criar_receita
        OnMouseClick: write the text variable via Default, min 0, max 300
    Rectangle (5,485 175x52), "P08 - (X,Y)", invisible if: Recipe_Pontos_Solda_Select<8
    Rectangle (195,485 105x52), "%s mm", text variable: Recipe_P_X08_Solda_Select, invisible if: Recipe_Pontos_Solda_Select<8, input disabled if: Not b_editar_receita and Not b_criar_receita
        OnMouseClick: write the text variable via Default, min 0, max 300
    Rectangle (5,545 175x52), "P09 - (X,Y)", invisible if: Recipe_Pontos_Solda_Select<9
    Rectangle (195,545 105x52), "%s mm", text variable: Recipe_P_X09_Solda_Select, invisible if: Recipe_Pontos_Solda_Select<9, input disabled if: Not b_editar_receita and Not b_criar_receita
        OnMouseClick: write the text variable via Default, min 0, max 300
    Rectangle (5,605 175x52), "P10 - (X,Y)", invisible if: Recipe_Pontos_Solda_Select<10
    Rectangle (195,605 105x52), "%s mm", text variable: Recipe_P_X10_Solda_Select, invisible if: Recipe_Pontos_Solda_Select<10, input disabled if: Not b_editar_receita and Not b_criar_receita
        OnMouseClick: write the text variable via Default, min 0, max 300
    Rectangle (302,365 105x52), "%s mm", text variable: Recipe_P_Y06_Solda_Select, invisible if: Recipe_Pontos_Solda_Select<6, input disabled if: Not b_editar_receita and Not b_criar_receita
        OnMouseClick: write the text variable via Default, min 0, max 300
    Rectangle (302,425 105x52), "%s mm", text variable: Recipe_P_Y07_Solda_Select, invisible if: Recipe_Pontos_Solda_Select<7, input disabled if: Not b_editar_receita and Not b_criar_receita
        OnMouseClick: write the text variable via Default, min 0, max 300
    Rectangle (302,485 105x52), "%s mm", text variable: Recipe_P_Y08_Solda_Select, invisible if: Recipe_Pontos_Solda_Select<8, input disabled if: Not b_editar_receita and Not b_criar_receita
        OnMouseClick: write the text variable via Default, min 0, max 300
    Rectangle (302,545 105x52), "%s mm", text variable: Recipe_P_Y09_Solda_Select, invisible if: Recipe_Pontos_Solda_Select<9, input disabled if: Not b_editar_receita and Not b_criar_receita
        OnMouseClick: write the text variable via Default, min 0, max 300
    Rectangle (302,605 105x52), "%s mm", text variable: Recipe_P_Y10_Solda_Select, invisible if: Recipe_Pontos_Solda_Select<10, input disabled if: Not b_editar_receita and Not b_criar_receita
        OnMouseClick: write the text variable via Default, min 0, max 300
    Checkbox (437,371 40x40), variable: Recipe_P06_Solda_Select, invisible if: Recipe_Pontos_Solda_Select<6, input disabled if: Not b_editar_receita and Not b_criar_receita
    Checkbox (437,431 40x40), variable: Recipe_P07_Solda_Select, invisible if: Recipe_Pontos_Solda_Select<7, input disabled if: Not b_editar_receita and Not b_criar_receita
    Checkbox (437,491 40x40), variable: Recipe_P08_Solda_Select, invisible if: Recipe_Pontos_Solda_Select<8, input disabled if: Not b_editar_receita and Not b_criar_receita
    Checkbox (437,551 40x40), variable: Recipe_P09_Solda_Select, invisible if: Recipe_Pontos_Solda_Select<9, input disabled if: Not b_editar_receita and Not b_criar_receita
    Checkbox (437,611 40x40), variable: Recipe_P10_Solda_Select, invisible if: Recipe_Pontos_Solda_Select<10, input disabled if: Not b_editar_receita and Not b_criar_receita
    Rectangle (5,665 175x52), "P11 - (X,Y)", invisible if: Recipe_Pontos_Solda_Select<11
    Rectangle (195,665 105x52), "%s mm", text variable: Recipe_P_X11_Solda_Select, invisible if: Recipe_Pontos_Solda_Select<11, input disabled if: Not b_editar_receita and Not b_criar_receita
        OnMouseClick: write the text variable via Default, min 0, max 300
    Rectangle (5,725 175x52), "P12 - (X,Y)", invisible if: Recipe_Pontos_Solda_Select<12
    Rectangle (195,725 105x52), "%s mm", text variable: Recipe_P_X12_Solda_Select, invisible if: Recipe_Pontos_Solda_Select<12, input disabled if: Not b_editar_receita and Not b_criar_receita
        OnMouseClick: write the text variable via Default, min 0, max 300
    Rectangle (302,665 105x52), "%s mm", text variable: Recipe_P_Y11_Solda_Select, invisible if: Recipe_Pontos_Solda_Select<11, input disabled if: Not b_editar_receita and Not b_criar_receita
        OnMouseClick: write the text variable via Default, min 0, max 300
    Rectangle (302,725 105x52), "%s mm", text variable: Recipe_P_Y12_Solda_Select, invisible if: Recipe_Pontos_Solda_Select<12, input disabled if: Not b_editar_receita and Not b_criar_receita
        OnMouseClick: write the text variable via Default, min 0, max 300
    Checkbox (437,671 40x40), variable: Recipe_P11_Solda_Select, invisible if: Recipe_Pontos_Solda_Select<11, input disabled if: Not b_editar_receita and Not b_criar_receita
    Checkbox (437,731 40x40), variable: Recipe_P12_Solda_Select, invisible if: Recipe_Pontos_Solda_Select<12, input disabled if: Not b_editar_receita and Not b_criar_receita
END_VISUALIZATION

// ---- VISUs/Lista_PontosRoboCamera.TcVIS
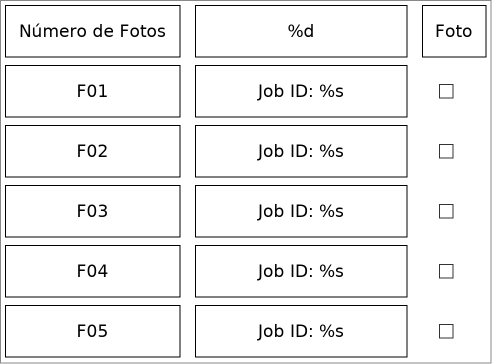
VISUALIZATION Lista_PontosRoboCamera  // 492x364
    Rectangle (5,5 175x52), "Número de Fotos"
    Rectangle (195,5 212x52), "%d", text variable: Recipe_Pontos_Camera_Select, input disabled if: Not b_editar_receita and Not b_criar_receita
        OnMouseClick: write the text variable via Default, min 0, max 5
    Rectangle (5,65 175x52), "F01", invisible if: Recipe_Pontos_Camera_Select<1
    Rectangle (195,65 212x52), "Job ID: %s", text variable: Recipe_JobID_F01_Camera_Select, invisible if: Recipe_Pontos_Camera_Select<1, input disabled if: Not b_editar_receita and Not b_criar_receita
        OnMouseClick: write the text variable via Default, min 0, max 500
    Rectangle (5,125 175x52), "F02", invisible if: Recipe_Pontos_Camera_Select<2
    Rectangle (195,125 212x52), "Job ID: %s", text variable: Recipe_JobID_F02_Camera_Select, invisible if: Recipe_Pontos_Camera_Select<2, input disabled if: Not b_editar_receita and Not b_criar_receita
        OnMouseClick: write the text variable via Default, min 0, max 500
    Rectangle (5,185 175x52), "F03", invisible if: Recipe_Pontos_Camera_Select<3
    Rectangle (195,185 212x52), "Job ID: %s", text variable: Recipe_JobID_F03_Camera_Select, invisible if: Recipe_Pontos_Camera_Select<3, input disabled if: Not b_editar_receita and Not b_criar_receita
        OnMouseClick: write the text variable via Default
    Rectangle (5,245 175x52), "F04", invisible if: Recipe_Pontos_Camera_Select<4
    Rectangle (195,245 212x52), "Job ID: %s", text variable: Recipe_JobID_F04_Camera_Select, invisible if: Recipe_Pontos_Camera_Select<4, input disabled if: Not b_editar_receita and Not b_criar_receita
        OnMouseClick: write the text variable via Default
    Rectangle (5,305 175x52), "F05", invisible if: Recipe_Pontos_Camera_Select<5
    Rectangle (195,305 212x52), "Job ID: %s", text variable: Recipe_JobID_F05_Camera_Select, invisible if: Recipe_Pontos_Camera_Select<5, input disabled if: Not b_editar_receita and Not b_criar_receita
        OnMouseClick: write the text variable via Default
    Rectangle (422,5 64x52), "Foto"
    Checkbox (437,71 40x40), variable: TRUE, invisible if: Recipe_Pontos_Camera_Select<1, input disabled if: TRUE
    Checkbox (437,131 40x40), variable: TRUE, invisible if: Recipe_Pontos_Camera_Select<2, input disabled if: TRUE
    Checkbox (437,191 40x40), variable: TRUE, invisible if: Recipe_Pontos_Camera_Select<3, input disabled if: TRUE
    Checkbox (437,251 40x40), variable: TRUE, invisible if: Recipe_Pontos_Camera_Select<4, input disabled if: TRUE
    Checkbox (437,311 40x40), variable: TRUE, invisible if: Recipe_Pontos_Camera_Select<5, input disabled if: TRUE
END_VISUALIZATION

// ---- VISUs/Tela_Alarmes_2.TcVIS
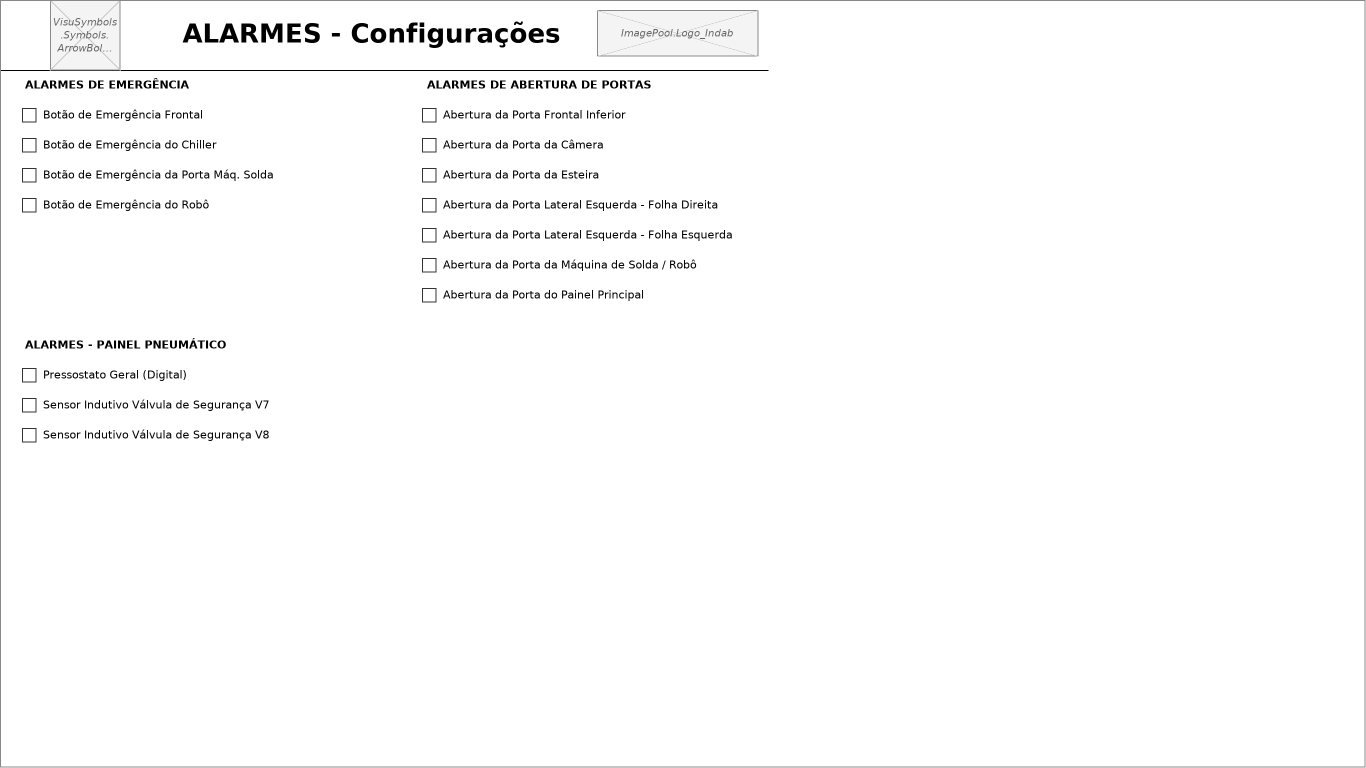
VISUALIZATION Tela_Alarmes_2  // 1366x768
    Line (0,70) (768,70)
    Line (0,1312) (768,1312)
    Image (597,10 161x46), image: ImagePool.Logo_Indab
    Rectangle (584,1340 180x24), "%t[dd/MM/yyyy]"
    Rectangle (584,1316 180x24), "%t[HH:mm:ss]"
    Label (153,7 437x53), "ALARMES - Configurações"
    Button (15,1315 175x45), "RECEITAS"
        OnMouseClick: change screen: Tela_Receita
    Checkbox (420,190 313x30), "Abertura da Porta Lateral Esquerda - Folha Direita"
    Checkbox (420,220 329x30), "Abertura da Porta Lateral Esquerda - Folha Esquerda"
    Checkbox (420,250 296x30), "Abertura da Porta da Máquina de Solda / Robô"
    Rectangle (22,75 237x20), "ALARMES DE EMERGÊNCIA"
    Rectangle (424,75 237x20), "ALARMES DE ABERTURA DE PORTAS"
    Checkbox (20,100 200x30), "Botão de Emergência Frontal"
    Checkbox (20,130 214x30), "Botão de Emergência do Chiller"
    Checkbox (20,160 278x30), "Botão de Emergência da Porta Máq. Solda"
    Checkbox (20,190 220x30), "Botão de Emergência do Robô"
    Checkbox (420,100 238x30), "Abertura da Porta Frontal Inferior"
    Checkbox (420,130 200x30), "Abertura da Porta da Câmera"
    Checkbox (420,160 200x30), "Abertura da Porta da Esteira"
    Checkbox (420,280 243x30), "Abertura da Porta do Painel Principal"
    Rectangle (22,335 237x20), "ALARMES - PAINEL PNEUMÁTICO"
    Checkbox (20,360 200x30), "Pressostato Geral (Digital)"
    Checkbox (20,390 286x30), "Sensor Indutivo Válvula de Segurança V7"
    Checkbox (20,420 278x30), "Sensor Indutivo Válvula de Segurança V8"
    Image (50,0 70x70), image: VisuSymbols.Symbols.ArrowBoldLeft
        OnMouseClick: change screen: Tela_Alarmes_1
    Button (375,1315 175x45), "PRODUÇÃO"
        OnMouseClick: change screen: Tela_Producao
    Button (195,1315 175x45), "MANUTENÇÃO"
        OnMouseClick: change screen: Tela_Manutencao
END_VISUALIZATION

// ---- VISUs/Tela_Manual_2.TcVIS
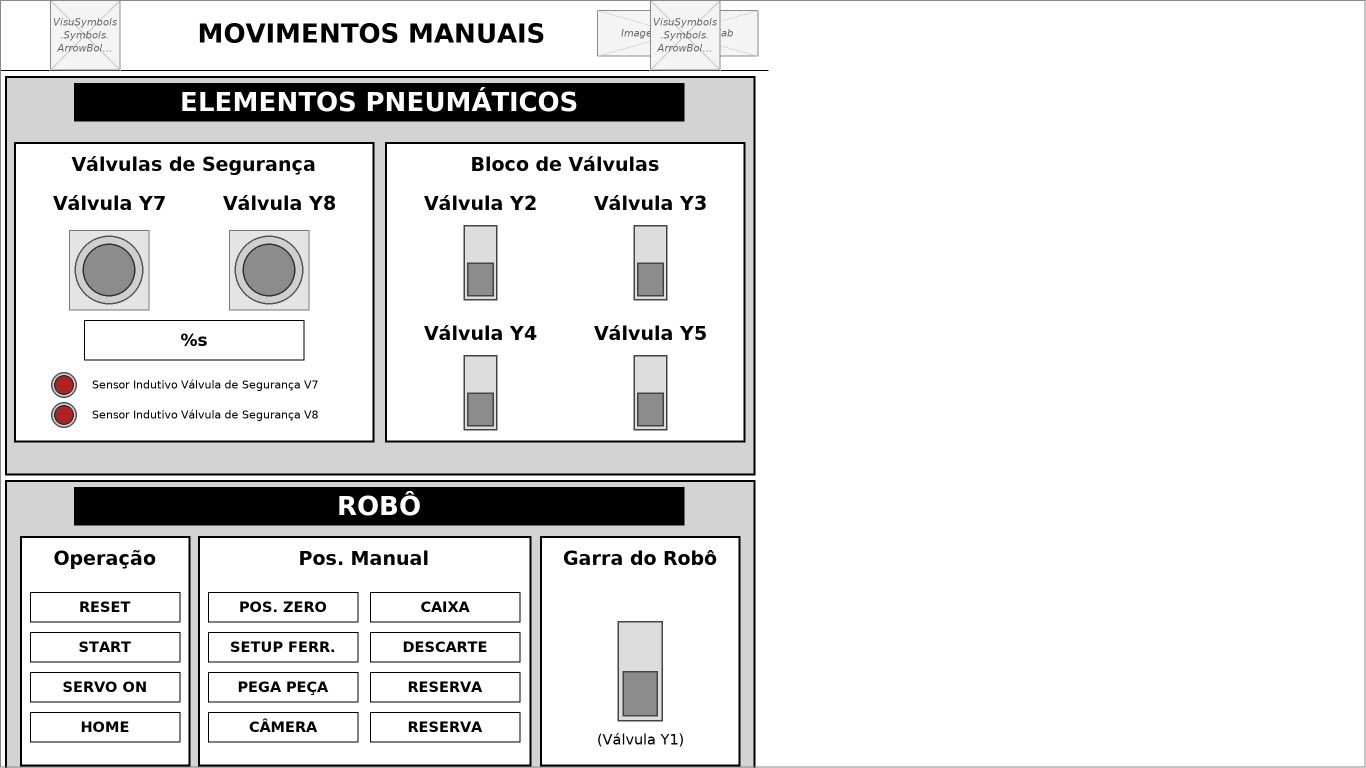
VISUALIZATION Tela_Manual_2  // 1366x768
    Group (5,480 750x305)
        RoundedRectangle (0,0 750x305)
        Rectangle (69,7 610x38), "ROBÔ", text variable: Recipe_name_Select, input disabled if: TRUE
        RoundedRectangle (15,56 170x230), input disabled if: TRUE
        Rectangle (20,65 160x27), "Operação", text variable: Recipe_name_Select, input disabled if: TRUE
        RoundedRectangle (25,112 150x30), "RESET", input disabled if: TRUE
            tap Servos.ResetServoX
        RoundedRectangle (25,152 150x30), "START", colour toggle: NOT Servos.PowerOnServoX, input disabled if: TRUE
        RoundedRectangle (193,56 333x230), input disabled if: TRUE
        Rectangle (279,65 160x27), "Pos. Manual", text variable: Recipe_name_Select, input disabled if: TRUE
        RoundedRectangle (203,112 150x30), "POS. ZERO", input disabled if: TRUE
        RoundedRectangle (203,152 150x30), "SETUP FERR.", colour toggle: NOT Servos.PowerOnServoX, input disabled if: TRUE
        RoundedRectangle (203,192 150x30), "PEGA PEÇA", colour toggle: NOT Servos.PowerOnServoX, input disabled if: TRUE
        RoundedRectangle (203,232 150x30), "CÂMERA", colour toggle: NOT Servos.PowerOnServoX, input disabled if: TRUE
        RoundedRectangle (535,56 200x230), input disabled if: TRUE
        Rectangle (545,65 180x27), "Garra do Robô", text variable: Recipe_name_Select, input disabled if: TRUE
        RoundedRectangle (25,232 150x30), "HOME", colour toggle: NOT Servos.PowerOnServoX, input disabled if: TRUE
        RoundedRectangle (25,192 150x30), "SERVO ON", input disabled if: TRUE
            tap Servos.ResetServoX
        DipSwitch (585,141 100x100), variable: IhmBt_Y1_Ligar, input disabled if: NOT MaquinaModoManual, behaviour: TOGGLE, style: Switch-DipSwitch-Gray
        Rectangle (578,246 115x27), "(Válvula Y1)", text variable: Recipe_name_Select, input disabled if: TRUE
        RoundedRectangle (365,232 150x30), "RESERVA", colour toggle: NOT Servos.PowerOnServoX, input disabled if: TRUE
        RoundedRectangle (365,112 150x30), "CAIXA", input disabled if: TRUE
        RoundedRectangle (365,152 150x30), "DESCARTE", colour toggle: NOT Servos.PowerOnServoX, input disabled if: TRUE
        RoundedRectangle (365,192 150x30), "RESERVA", colour toggle: NOT Servos.PowerOnServoX, input disabled if: TRUE
    Line (0,70) (768,70)
    Line (0,1312) (768,1312)
    Image (597,10 161x46), image: ImagePool.Logo_Indab
    Rectangle (584,1340 180x24), "%t[dd/MM/yyyy]"
    Rectangle (584,1316 180x24), "%t[HH:mm:ss]"
    Label (153,7 437x53), "MOVIMENTOS MANUAIS"
    Button (15,1315 175x45), "RECEITAS"
        OnMouseClick: change screen: Tela_Receita
    Button (375,1315 175x45), "MANUTENÇÃO"
        OnMouseClick: change screen: Tela_Manutencao
    Image (50,0 70x70), image: VisuSymbols.Symbols.ArrowBoldLeft
        OnMouseClick: change screen: Tela_Manual_1
    Image (650,0 70x70), image: VisuSymbols.Symbols.ArrowBoldRight
        OnMouseClick: change screen: Tela_Manual_3
    Button (195,1315 175x45), "PRODUÇÃO"
        OnMouseClick: change screen: Tela_Producao
    RoundedRectangle (5,76 750x399)
    Rectangle (74,83 610x38), "ELEMENTOS PNEUMÁTICOS", text variable: Recipe_name_Select
    RoundedRectangle (385,142 360x300), input disabled if: NOT MaquinaModoManual
    Rectangle (399,151 332x27), "Bloco de Válvulas", text variable: Recipe_name_Select, input disabled if: NOT MaquinaModoManual
    RoundedRectangle (14,142 360x300), input disabled if: NOT MaquinaModoManual
    Rectangle (28,151 332x27), "Válvulas de Segurança", text variable: Recipe_name_Select, input disabled if: NOT MaquinaModoManual
    Rectangle (52,190 115x27), "Válvula Y7", text variable: Recipe_name_Select, input disabled if: TRUE
    Rectangle (222,190 115x27), "Válvula Y8", text variable: Recipe_name_Select, input disabled if: TRUE
    PushSwitchLed (69,230 80x80), variable: IhmBt_Y7_Ligar, input disabled if: TRUE, behaviour: TOGGLE, style: Switch-PushSwitchLed-Gray
    PushSwitchLed (229,230 80x80), variable: IhmBt_Y8_Ligar, input disabled if: TRUE, behaviour: TOGGLE, style: Switch-PushSwitchLed-Gray
    Rectangle (423,190 115x27), "Válvula Y2", text variable: Recipe_name_Select, input disabled if: NOT MaquinaModoManual
    Rectangle (593,190 115x27), "Válvula Y3", text variable: Recipe_name_Select, input disabled if: NOT MaquinaModoManual
    DipSwitch (443,225 75x75), variable: IhmBt_Y2_Ligar, input disabled if: NOT MaquinaModoManual, behaviour: TOGGLE, style: Switch-DipSwitch-Gray
    DipSwitch (613,225 75x75), variable: IhmBt_Y3_Ligar, input disabled if: NOT MaquinaModoManual, behaviour: TOGGLE, style: Switch-DipSwitch-Gray
    Rectangle (423,320 115x27), "Válvula Y4", text variable: Recipe_name_Select, input disabled if: NOT MaquinaModoManual
    Rectangle (593,320 115x27), "Válvula Y5", text variable: Recipe_name_Select, input disabled if: NOT MaquinaModoManual
    DipSwitch (613,355 75x75), variable: IhmBt_Y5_Ligar, input disabled if: NOT MaquinaModoManual, behaviour: TOGGLE, style: Switch-DipSwitch-Gray
    DipSwitch (443,355 75x75), variable: IhmBt_Y4_Ligar, input disabled if: NOT MaquinaModoManual, behaviour: TOGGLE, style: Switch-DipSwitch-Gray
    Rectangle (84,320 220x40), "%s", text variable: IhmVs_PressaoPainelPneumatico_Text, colour toggle: Alarmes.ByteAlarmePainelPneumatico.0, input disabled if: NOT MaquinaModoManual
    Group (49,370 290x60), input disabled if: NOT MaquinaModoManual
        Rectangle (40,30 250x30), "Sensor Indutivo Válvula de Segurança V8"
        Lamp1 (0,0 30x30), variable: Alarmes.ByteAlarmePainelPneumatico.1, style: Lamp-Lamp1-Red
        Rectangle (40,0 250x30), "Sensor Indutivo Válvula de Segurança V7"
        Lamp1 (0,30 30x30), variable: Alarmes.ByteAlarmePainelPneumatico.2, style: Lamp-Lamp1-Red
    Line (-1,1315) (767,1315)
    RoundedRectangle (5,790 750x511)
    Rectangle (75,800 610x38), "MOTORES", text variable: Recipe_name_Select, input disabled if: NOT MaquinaModoManual
    Button (260,1235 240x60), "MODO: %s", text variable: IhmBt_ManualAuto_Text, colour toggle: IhmBt_ManualAuto_Color
        toggle IhmBt_ManualAuto
    RoundedRectangle (24,855 350x360), input disabled if: NOT MaquinaModoManual
    Rectangle (146,863 106x27), "Servo X", text variable: Recipe_name_Select, input disabled if: NOT MaquinaModoManual
    Rectangle (31,895 77x22), "Posição", input disabled if: NOT MaquinaModoManual
    Rectangle (106,895 90x22), "%.2f mm", text variable: IhmLeit_ServoX_Posicao, input disabled if: NOT MaquinaModoManual
    RoundedRectangle (38,1165 150x30), "REFERENCIAR", input disabled if: NOT MaquinaModoManual
        tap IhmBt_ServoX_Referenciar
    RoundedRectangle (38,1125 150x30), "POWER ON", input disabled if: NOT MaquinaModoManual
        toggle IhmBt_ServoX_PowerOn
    RoundedRectangle (38,1025 150x30), "HOME", colour toggle: NOT Servos.PowerOnServoX, input disabled if: NOT MaquinaModoManual
        tap IhmBt_ServoX_Home
    RoundedRectangle (38,985 150x30), "RESET", input disabled if: NOT MaquinaModoManual
        tap IhmBt_ServoX_Reset
    Image (38,1065 50x50), invisible if: NOT IhmBt_ServoX_PowerOn, input disabled if: NOT MaquinaModoManual, image: VisuSymbols.Symbols.ArrowBoldLeft
        OnMouseDown: execute { IhmBt_ServoX_JogBwd := TRUE; }
        OnMouseLeave: execute { IhmBt_ServoX_JogBwd := FALSE; }
        OnMouseUp: execute { IhmBt_ServoX_JogBwd := FALSE; }
    Image (138,1065 50x50), invisible if: NOT IhmBt_ServoX_PowerOn, input disabled if: NOT MaquinaModoManual, image: VisuSymbols.Symbols.ArrowBoldRight
        OnMouseDown: execute { IhmBt_ServoX_JogFwd := TRUE; }
        OnMouseLeave: execute { IhmBt_ServoX_JogFwd := FALSE; }
        OnMouseUp: execute { IhmBt_ServoX_JogFwd := FALSE; }
    Rectangle (90,1079 45x20), "JOG", invisible if: NOT IhmBt_ServoX_PowerOn, input disabled if: NOT MaquinaModoManual
    Rectangle (31,920 77x22), "Velocidade:", input disabled if: NOT MaquinaModoManual
    Rectangle (106,920 90x22), "%.2f mm/s", text variable: IhmLeit_ServoX_Velocidade, input disabled if: NOT MaquinaModoManual
    Rectangle (31,945 77x22), "Torque:", input disabled if: NOT MaquinaModoManual
    Rectangle (106,945 90x22), "%d kgfm", text variable: IhmLeit_ServoX_Torque, input disabled if: NOT MaquinaModoManual
    RoundedRectangle (384,855 350x360), input disabled if: NOT MaquinaModoManual
    Rectangle (506,864 106x27), "Servo Y", text variable: Recipe_name_Select, input disabled if: NOT MaquinaModoManual
    RoundedRectangle (398,1165 150x30), "REFERENCIAR", input disabled if: NOT MaquinaModoManual
        tap IhmBt_ServoY_Referenciar
    RoundedRectangle (398,1125 150x30), "POWER ON", input disabled if: NOT MaquinaModoManual
        toggle IhmBt_ServoY_PowerOn
    RoundedRectangle (398,1025 150x30), "HOME", colour toggle: NOT Servos.PowerOnServoX, input disabled if: NOT MaquinaModoManual
        tap IhmBt_ServoY_Home
    RoundedRectangle (398,985 150x30), "RESET", input disabled if: NOT MaquinaModoManual
        tap IhmBt_ServoY_Reset
    Image (398,1065 50x50), invisible if: NOT IhmBt_ServoY_PowerOn, input disabled if: NOT MaquinaModoManual, image: VisuSymbols.Symbols.ArrowBoldLeft
        OnMouseDown: execute { IhmBt_ServoY_JogBwd := TRUE; }
        OnMouseLeave: execute { IhmBt_ServoY_JogBwd := FALSE; }
        OnMouseUp: execute { IhmBt_ServoY_JogBwd := FALSE; }
    Image (498,1065 50x50), invisible if: NOT IhmBt_ServoY_PowerOn, input disabled if: NOT MaquinaModoManual, image: VisuSymbols.Symbols.ArrowBoldRight
        OnMouseDown: execute { IhmBt_ServoY_JogFwd := TRUE; }
        OnMouseLeave: execute { IhmBt_ServoY_JogFwd := FALSE; }
        OnMouseUp: execute { IhmBt_ServoY_JogFwd := FALSE; }
    Rectangle (450,1079 45x20), "JOG", text variable: Recipe_name_Select, invisible if: NOT IhmBt_ServoY_PowerOn, input disabled if: NOT MaquinaModoManual
    Rectangle (391,895 77x22), "Posição", input disabled if: NOT MaquinaModoManual
    Rectangle (391,920 77x22), "Velocidade:", input disabled if: NOT MaquinaModoManual
    Rectangle (391,945 77x22), "Torque:", input disabled if: NOT MaquinaModoManual
    Rectangle (466,945 90x22), "%d kgfm", text variable: IhmLeit_ServoY_Torque, input disabled if: NOT MaquinaModoManual
    Rectangle (466,895 90x22), "%.2f mm", text variable: IhmLeit_ServoY_Posicao, input disabled if: NOT MaquinaModoManual
    Rectangle (466,920 90x22), "%.2f mm/s", text variable: IhmLeit_ServoY_Velocidade, input disabled if: NOT MaquinaModoManual
    RoundedRectangle (210,915 150x30), "INICIO DE CURSO", input disabled if: MaquinaModoAuto OR NOT IhmBt_ServoX_PowerOn
        toggle IhmBt_ServoX_ReferenciarAutoINICIO
    Rectangle (220,1125 130x30), "(Sensor Fim de Curso)"
    Lamp1 (270,955 30x30), variable: InFimCurso3, style: Lamp-Lamp1-Red
    Rectangle (220,985 130x30), "(Sensor Fim de Curso)"
    Lamp1 (270,1095 30x30), variable: InFimCurso4, style: Lamp-Lamp1-Red
    RoundedRectangle (210,1055 150x30), "FIM DE CURSO", input disabled if: MaquinaModoAuto OR NOT IhmBt_ServoX_PowerOn
        toggle IhmBt_ServoX_ReferenciarAutoFIM
    RoundedRectangle (570,915 150x30), "INICIO DE CURSO", input disabled if: MaquinaModoAuto OR NOT IhmBt_ServoY_PowerOn
        toggle IhmBt_ServoY_ReferenciarAutoINICIO
    Lamp1 (630,955 30x30), variable: InFimCurso1, style: Lamp-Lamp1-Red
    Rectangle (580,1125 130x30), "(Sensor Fim de Curso)"
    Rectangle (580,985 130x30), "(Sensor Fim de Curso)"
    Lamp1 (630,1095 30x30), variable: InFimCurso2, style: Lamp-Lamp1-Red
    RoundedRectangle (570,1055 150x30), "FIM DE CURSO", input disabled if: MaquinaModoAuto OR NOT IhmBt_ServoY_PowerOn
        toggle IhmBt_ServoY_ReferenciarAutoFIM
END_VISUALIZATION

// ---- VISUs/Tela_Manual_3.TcVIS
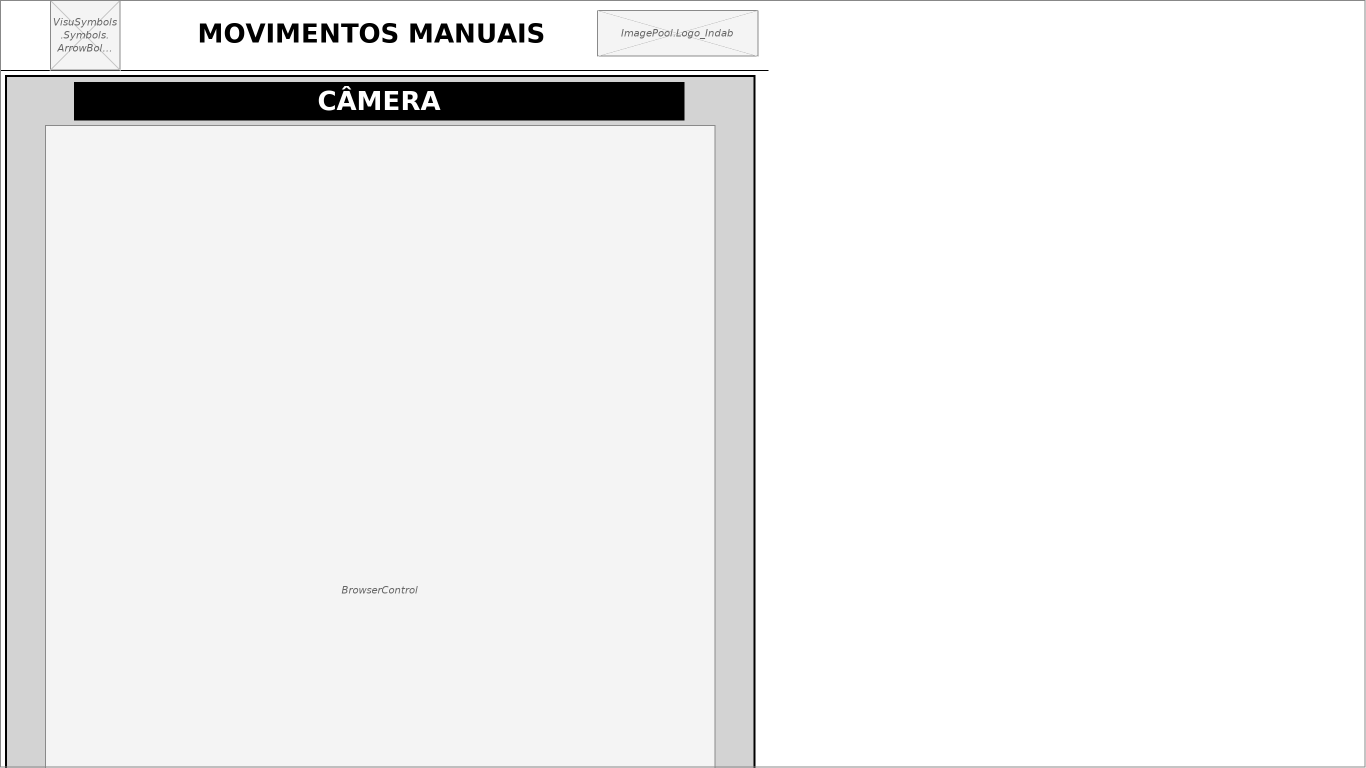
VISUALIZATION Tela_Manual_3  // 1366x768
    Line (0,70) (768,70)
    Line (0,1312) (768,1312)
    Image (597,10 161x46), image: ImagePool.Logo_Indab
    Rectangle (584,1340 180x24), "%t[dd/MM/yyyy]"
    Rectangle (584,1316 180x24), "%t[HH:mm:ss]"
    Label (153,7 437x53), "MOVIMENTOS MANUAIS"
    Button (15,1315 175x45), "RECEITAS"
        OnMouseClick: change screen: Tela_Receita
    Button (375,1315 175x45), "MANUTENÇÃO"
        OnMouseClick: change screen: Tela_Manutencao
    RoundedRectangle (5,75 750x1230)
    Rectangle (74,82 610x38), "CÂMERA", text variable: Recipe_name_Select
    Image (50,0 70x70), image: VisuSymbols.Symbols.ArrowBoldLeft
        OnMouseClick: change screen: Tela_Manual_2
    BrowserControl (45,125 670x930)
        p3734058945: MAIN.sUrlAddressCamera
    Button (195,1315 175x45), "PRODUÇÃO"
        OnMouseClick: change screen: Tela_Producao
    RoundedRectangle (207,1180 150x30), "TRIGGER", input disabled if: NOT MaquinaModoManual
        tap IhmBt_Camera_Trigger
    Rectangle (226,1110 130x25), "ID: %d", text variable: IhmEscr_Camera_SetJob
        OnMouseClick: write the text variable via Default, min 0, max 300
    Rectangle (50,1113 155x20), "Selecionar Job (Job ID):", input disabled if: NOT MaquinaModoManual
    Rectangle (226,1140 130x25), "%.2f s", text variable: IhmEscr_Camera_DelayError
        OnMouseClick: write the text variable via Default, min 0, max 300
    Rectangle (50,1143 130x20), "Delay (ERROR):", input disabled if: NOT MaquinaModoManual
    Rectangle (447,1115 180x22), "Executando Job (Job ID):", input disabled if: NOT MaquinaModoManual
    Rectangle (500,1070 180x27), "Status Câmera", text variable: Recipe_name_Select, input disabled if: NOT MaquinaModoManual
    Rectangle (623,1115 90x22), "%d", text variable: IhmLeit_Camera_JobID, input disabled if: NOT MaquinaModoManual
    Rectangle (109,1070 188x27), "Controle Manual:", text variable: Recipe_name_Select, input disabled if: NOT MaquinaModoManual
    Button (260,1235 240x60), "MODO: %s", text variable: IhmBt_ManualAuto_Text, colour toggle: IhmBt_ManualAuto_Color
        toggle IhmBt_ManualAuto
    RoundedRectangle (50,1180 150x30), "CHANGE JOG", input disabled if: NOT MaquinaModoManual
        tap IhmBt_Camera_ChangeJob
    Rectangle (619,1181 100x30), "%s", colour toggle: IhmLed_Camera_JobResult, input disabled if: NOT MaquinaModoManual
    Lamp1 (653,1146 30x30), variable: IhmLed_Camera_JobCompleted, style: Lamp-Lamp1-Red
    Rectangle (447,1150 180x22), "Job Completed:", input disabled if: NOT MaquinaModoManual
    Rectangle (447,1185 180x22), "Job Result:", input disabled if: NOT MaquinaModoManual
END_VISUALIZATION

// ---- VISUs/Tela_Alarmes_1.TcVIS
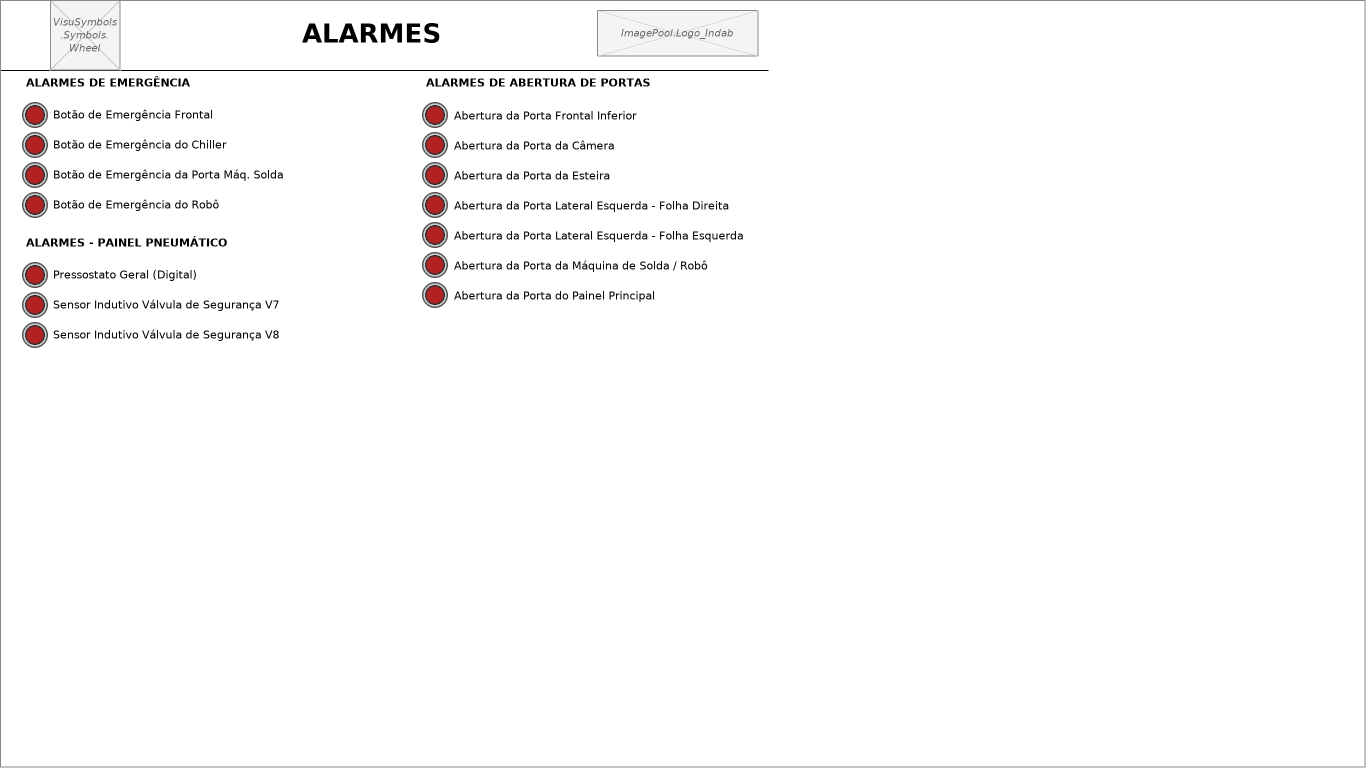
VISUALIZATION Tela_Alarmes_1  // 1366x768
    Line (0,70) (768,70)
    Line (0,1312) (768,1312)
    Image (597,10 161x46), image: ImagePool.Logo_Indab
    Rectangle (584,1340 180x24), "%t[dd/MM/yyyy]"
    Rectangle (584,1316 180x24), "%t[HH:mm:ss]"
    Label (153,7 437x53), "ALARMES"
    Lamp1 (20,100 30x30), variable: Alarmes.ByteAlarmeEmergencia.0, style: Lamp-Lamp1-Red
    Rectangle (50,100 250x30), "Botão de Emergência Frontal"
    Lamp1 (20,130 30x30), variable: Alarmes.ByteAlarmeEmergencia.1, style: Lamp-Lamp1-Red
    Rectangle (50,130 250x30), "Botão de Emergência do Chiller"
    Lamp1 (20,160 30x30), variable: Alarmes.ByteAlarmeEmergencia.2, style: Lamp-Lamp1-Red
    Rectangle (50,160 250x30), "Botão de Emergência da Porta Máq. Solda"
    Lamp1 (20,190 30x30), variable: Alarmes.ByteAlarmeEmergencia.3, style: Lamp-Lamp1-Red
    Rectangle (50,190 250x30), "Botão de Emergência do Robô"
    Rectangle (23,73 237x20), "ALARMES DE EMERGÊNCIA"
    Lamp1 (420,100 30x30), variable: Alarmes.ByteAlarmeAberturaPortas.0, style: Lamp-Lamp1-Red
    Rectangle (451,101 300x30), "Abertura da Porta Frontal Inferior"
    Lamp1 (420,130 30x30), variable: Alarmes.ByteAlarmeAberturaPortas.1, style: Lamp-Lamp1-Red
    Rectangle (451,131 300x30), "Abertura da Porta da Câmera"
    Lamp1 (420,160 30x30), variable: Alarmes.ByteAlarmeAberturaPortas.2, style: Lamp-Lamp1-Red
    Rectangle (451,161 300x30), "Abertura da Porta da Esteira"
    Lamp1 (420,190 30x30), variable: Alarmes.ByteAlarmeAberturaPortas.3, style: Lamp-Lamp1-Red
    Rectangle (451,191 300x30), "Abertura da Porta Lateral Esquerda - Folha Direita"
    Lamp1 (420,220 30x30), variable: Alarmes.ByteAlarmeAberturaPortas.4, style: Lamp-Lamp1-Red
    Rectangle (451,221 300x30), "Abertura da Porta Lateral Esquerda - Folha Esquerda"
    Lamp1 (420,250 30x30), variable: Alarmes.ByteAlarmeAberturaPortas.5, style: Lamp-Lamp1-Red
    Rectangle (451,251 300x30), "Abertura da Porta da Máquina de Solda / Robô"
    Lamp1 (420,280 30x30), variable: Alarmes.ByteAlarmeAberturaPortas.6, style: Lamp-Lamp1-Red
    Rectangle (451,281 300x30), "Abertura da Porta do Painel Principal"
    Rectangle (423,73 237x20), "ALARMES DE ABERTURA DE PORTAS"
    Button (15,1315 175x45), "RECEITAS"
        OnMouseClick: change screen: Tela_Receita
    Lamp1 (20,260 30x30), variable: Alarmes.ByteAlarmePainelPneumatico.0, style: Lamp-Lamp1-Red
    Rectangle (50,260 250x30), "Pressostato Geral (Digital)"
    Lamp1 (20,290 30x30), variable: Alarmes.ByteAlarmePainelPneumatico.1, style: Lamp-Lamp1-Red
    Rectangle (50,290 250x30), "Sensor Indutivo Válvula de Segurança V7"
    Lamp1 (20,320 30x30), variable: Alarmes.ByteAlarmePainelPneumatico.2, style: Lamp-Lamp1-Red
    Rectangle (50,320 250x30), "Sensor Indutivo Válvula de Segurança V8"
    Rectangle (23,233 237x20), "ALARMES - PAINEL PNEUMÁTICO"
    Image (50,0 70x70), image: VisuSymbols.Symbols.Wheel
        OnMouseClick: change screen: Tela_Alarmes_2
    Button (375,1315 175x45), "PRODUÇÃO"
        OnMouseClick: change screen: Tela_Producao
    Button (195,1315 175x45), "MANUTENÇÃO"
        OnMouseClick: change screen: Tela_Manutencao
END_VISUALIZATION

// ---- VISUs/Tela_Producao.TcVIS
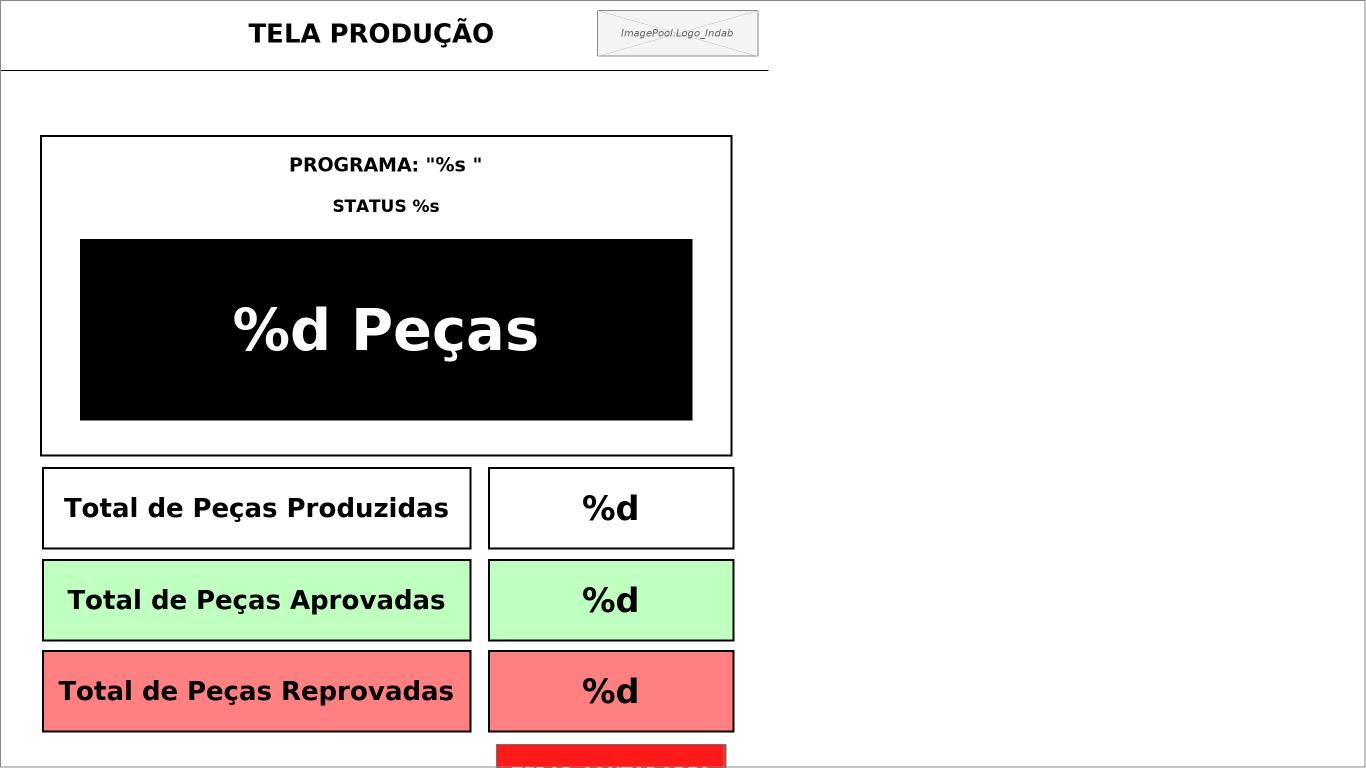
VISUALIZATION Tela_Producao  // 1366x768
    Line (0,1312) (768,1312)
    Rectangle (584,1340 180x24), "%t[dd/MM/yyyy]"
    Rectangle (584,1316 180x24), "%t[HH:mm:ss]"
    Group (0,7 768x64)
        Line (0,63) (768,63)
        Image (597,3 161x46), image: ImagePool.Logo_Indab
        Label (153,0 437x53), "TELA PRODUÇÃO"
    RoundedRectangle (40,135 692x321)
    RoundedRectangle (80,239 612x181), "%d Peças", text variable: Contador_Total
    Rectangle (81,147 610x36), "PROGRAMA: "%s "", text variable: Recipe_name_Select
    RoundedRectangle (42,467 429x82), "Total de Peças Produzidas"
    RoundedRectangle (488,467 246x82), "%d", text variable: Contador_Total
    RoundedRectangle (42,559 429x82), "Total de Peças Aprovadas"
    RoundedRectangle (488,559 246x82), "%d", text variable: Contador_PecasAprovadas
    RoundedRectangle (42,650 429x82), "Total de Peças Reprovadas"
    RoundedRectangle (488,650 246x82), "%d", text variable: Contador_PecasReprovadas
    RoundedRectangle (40,901 692x400)
    Button (496,744 230x60), "ZERAR CONTADORES"
        OnMouseClick: execute { BT_ihm_zerar_contador := TRUE; }
    Rectangle (80,925 610x35), "COMANDOS", text variable: Recipe_name_Select
    Button (15,1315 175x45), "RECEITAS"
        OnMouseClick: change screen: Tela_Receita
    Button (195,1315 175x45), "MANUTENÇÃO"
        OnMouseClick: change screen: Tela_Manutencao
    Rectangle (81,188 610x36), "STATUS %s"
    Button (375,1315 175x45), "ALARMES"
        OnMouseClick: change screen: Tela_Alarmes_1
    PowerSwitch (515,1075 143x136), variable: IhmBt_Desligar, behaviour: TOGGLE, style: Switch-PowerSwitch-Red
    PushSwitch (123,1034 90x90), variable: IhmBt_Ligar, behaviour: TOGGLE, style: Switch-PushSwitch-Green
    Rectangle (115,1000 106x38), "START", text variable: Recipe_name_Select
    PushSwitch (123,1184 90x90), variable: IhmBt_Reset, behaviour: TAP, style: Switch-PushSwitch-Blue
    Rectangle (115,1150 106x38), "RESET", text variable: Recipe_name_Select
    PushSwitch (323,1034 90x90), variable: IhmBt_Pausar, behaviour: TOGGLE, style: Switch-PushSwitch-Yellow
    Rectangle (315,1000 106x38), "PAUSE", text variable: Recipe_name_Select
    Rectangle (538,1031 106x38), "STOP", text variable: Recipe_name_Select
    Rectangle (278,1150 180x38), "COND. INICIAIS", text variable: Recipe_name_Select
    PushSwitch (323,1184 90x90), variable: IhmBt_CondIniciais, behaviour: TOGGLE, style: Switch-PushSwitch-Yellow
    Image (630,900 100x100), invisible if: NOT MaquinaAlarme, image: VisuSymbols.Symbols.Caution
    Button (496,810 230x60), "MODO: %s", text variable: IhmBt_ManualAuto_Text, colour toggle: IhmBt_ManualAuto_Color
        toggle IhmBt_ManualAuto
END_VISUALIZATION

